fbADSREAD(			PORT						:= 500, 
					IDXGRP						:= udiIDXGRP_OFFS + nAxisID, 
					IDXOFFS						:= nOffset, 
					LEN							:= 2, 
					DESTADDR					:= ADR(wData), 
					READ						:= bExecute, 
					BUSY						=> Out.Busy, 
					ERR							=> Out.Error, 
					ERRID						=> Out.ErrorID);

// Fix library issue, one extra cycle + Done
CASE nStep OF
	
	0: 
	
		Out.Error 								:= FALSE;
		Out.ErrorID 							:= 0;

		IF Out.Busy THEN
			nStep								:= nStep + 10;
		END_IF
	
	10:
	
		IF NOT Out.Busy THEN
			Out.Busy							:= TRUE;
			IF Out.Error THEN
				Out.ErrorID						:= 0;
				Out.Error						:= FALSE;
				nStep							:= 1000;
			ELSE
				nStep							:= 100;
			END_IF
		END_IF
		
	100, 1000:

		Out.Done								:= nStep = 100;
		Out.Error								:= nStep = 1000;
		IF Out.Error THEN
			Message := CONCAT('FB_NcSWLimitSwitchCtrl method ReadBool failed - Error ID: ',UDINT_TO_STRING(Out.ErrorID));
			Message := CONCAT(Message, '! FB instance: %s');
			ADSLOGSTR(ADSLOG_MSGTYPE_WARN,Message,sInstancePath);
		END_IF
		
		IF bExecute THEN
			nStep								:= nStep + 1;
		ELSE
			fbADSREAD(	READ					:= FALSE);
			nStep								:= 0;
		END_IF
		
	101, 1001:
	
		Out.Done								:= nStep = 101;
		Out.Error								:= nStep = 1001;
		IF NOT bExecute THEN
			fbADSREAD(	READ					:= FALSE);
			Out.Done							:= FALSE;
			Out.Error							:= FALSE;
			Out.ErrorID							:= 0;
			nStep								:= 0;
		END_IF	

END_CASE

pRead											:= Out;

bOut											:= wData.0;
ReadBool										:= Out;
END_METHOD

METHOD ReadLreal 								: Tc2_MC2.ST_McOutputs
VAR_INPUT
	bExecute									: BOOL;
	nAxisID										: UDINT;
	nOffset										: UDINT;
END_VAR
VAR_OUTPUT
	lrOut										: LREAL;
END_VAR
VAR_INST
	fbADSREAD									: ADSREAD;
	lrData										: LREAL;
	nStep										: DINT;
END_VAR
VAR
	Out											: Tc2_MC2.ST_McOutputs;
	Message										: STRING;
END_VAR
IF nAxisID = 0 THEN
	
	IF NOT bAxisIdError THEN
		ADSLOGSTR(ADSLOG_MSGTYPE_ERROR,'FB_NcSWLimitSwitchCtrl critical error - Axis ID not assigned! FB instance: %s',sInstancePath);
	END_IF
	
	bAxisIdError 								:= TRUE;
	RETURN;	
END_IF

fbADSREAD(			PORT						:= 500, 
					IDXGRP						:= udiIDXGRP_OFFS + nAxisID, 
					IDXOFFS						:= nOffset, 
					LEN							:= 8, 
					DESTADDR					:= ADR(lrData), 
					READ						:= bExecute, 
					BUSY						=> Out.Busy, 
					ERR							=> Out.Error, 
					ERRID						=> Out.ErrorID);

// Fix library issue, one extra cycle + Done
CASE nStep OF
	
	0: 
	
		Out.Error 								:= FALSE;
		Out.ErrorID 							:= 0;

		IF Out.Busy THEN
			nStep								:= nStep + 10;
		END_IF
	
	10:
	
		IF NOT Out.Busy THEN
			Out.Busy							:= TRUE;
			IF Out.Error THEN
				Out.ErrorID						:= 0;
				Out.Error						:= FALSE;
				nStep							:= 1000;
			ELSE
				nStep							:= 100;
			END_IF
		END_IF
		
	100, 1000:

		Out.Done								:= nStep = 100;
		Out.Error								:= nStep = 1000;
		IF Out.Error THEN
			Message := CONCAT('FB_NcSWLimitSwitchCtrl method ReadLreal failed - Error ID: ',UDINT_TO_STRING(Out.ErrorID));
			Message := CONCAT(Message, '! FB instance: %s');
			ADSLOGSTR(ADSLOG_MSGTYPE_WARN,Message,sInstancePath);
		END_IF
		
		IF bExecute THEN
			nStep								:= nStep + 1;
		ELSE
			fbADSREAD(	READ					:= FALSE);
			nStep								:= 0;
		END_IF
		
	101, 1001:
	
		Out.Done								:= nStep = 101;
		Out.Error								:= nStep = 1001;
		IF NOT bExecute THEN
			fbADSREAD(	READ					:= FALSE);
			Out.Done							:= FALSE;
			Out.Error							:= FALSE;
			Out.ErrorID							:= 0;
			nStep								:= 0;
		END_IF	

END_CASE

pRead											:= Out;

lrOut											:= lrData;
ReadLreal										:= Out;
END_METHOD

METHOD ReadParams 								: Tc2_MC2.ST_McOutputs
VAR_INPUT
	bExecute									: BOOL;
	nAxisID										: UDINT;
END_VAR
VAR_INST
	stOut	 									: Tc2_MC2.ST_McOutputs;
	nStep										: DINT;
END_VAR
VAR
	Out	 										: Tc2_MC2.ST_McOutputs;
END_VAR
CASE nStep OF

	0: 
		IF bExecute THEN
			stOut.Busy							:= TRUE;
			nStep								:= nStep + 5;
		END_IF
		
	5:

		Out 									:= ReadValueMin(bExecute := TRUE, nAxisID := nAxisID);
		IF Out.Busy THEN
			nStep								:= nStep + 5;
		END_IF
	
	10:
	
		Out 									:= ReadValueMin(bExecute := FALSE, nAxisID := nAxisID);
		IF Out.Done THEN
			nStep								:= nStep + 5;
		ELSIF Out.Error THEN
			nStep								:= 1000;
		END_IF
	
	15: 
	
		Out 									:= ReadValueMax(bExecute := TRUE, nAxisID := nAxisID);
		IF Out.Busy THEN
			nStep								:= nStep + 5;
		END_IF
		
	20:
	
		Out 									:= ReadValueMax(bExecute := FALSE, nAxisID := nAxisID);
		IF Out.Done THEN
			nStep								:= nStep + 5;
		ELSIF Out.Error THEN
			nStep								:= 1000;
		END_IF
	
	25: 
	
		Out 									:= ReadStateMin(bExecute := TRUE, nAxisID := nAxisID);
		IF Out.Busy THEN
			nStep								:= nStep + 5;
		END_IF
		
	30:
	
		Out 									:= ReadStateMin(bExecute := FALSE, nAxisID := nAxisID);
		IF Out.Done THEN
			nStep								:= nStep + 5;
		ELSIF Out.Error THEN
			nStep								:= 1000;
		END_IF
	
	35: 
	
		Out 									:= ReadStateMax(bExecute := TRUE, nAxisID := nAxisID);
		IF Out.Busy THEN
			nStep								:= nStep + 5;
		END_IF
		
	40:
	
		Out 									:= ReadStateMax(bExecute := FALSE, nAxisID := nAxisID);
		IF Out.Done THEN
			nStep								:= 100;
		ELSIF Out.Error THEN
			nStep								:= 1000;
		END_IF
		
	100, 1000:

		stOut.Busy								:= FALSE;
		stOut.Done								:= nStep = 100;
		stOut.Error								:= nStep = 1000;
		nStep									:= nStep + 1;
		
	101, 1001:
	
		IF NOT bExecute THEN
			stOut.Busy							:= FALSE;
			stOut.Done							:= FALSE;
			stOut.Error							:= FALSE;
			nStep								:= 0;			
		END_IF

END_CASE

ReadParams										:= stOut;
END_METHOD

METHOD ReadStateMax 							: Tc2_MC2.ST_McOutputs
VAR_INPUT
	bExecute									: BOOL;
	nAxisID										: UDINT;
END_VAR
VAR
	bOut										: BOOL;
END_VAR
ReadStateMax 									:= ReadBool(	bExecute 	:= bExecute, 
																nAxisID 	:= nAxisID, 
																nOffset 	:= 16#0000_000C, 
																bOut 		=> bOut);

LimitSwitchStateMax								:= bOut;
END_METHOD

METHOD ReadStateMin 							: Tc2_MC2.ST_McOutputs
VAR_INPUT
	bExecute									: BOOL;
	nAxisID										: UDINT;
END_VAR
VAR
	bOut										: BOOL;
END_VAR
ReadStateMin 									:= ReadBool(	bExecute 	:= bExecute, 
																nAxisID 	:= nAxisID, 
																nOffset 	:= 16#0000_000B, 
																bOut 		=> bOut);
																
LimitSwitchStateMin								:= bOut;
END_METHOD

METHOD ReadValueMax 							: Tc2_MC2.ST_McOutputs
VAR_INPUT
	bExecute									: BOOL;
	nAxisID										: UDINT;
END_VAR
VAR
	lrOut										: LREAL;
END_VAR
ReadValueMax 									:= ReadLreal(	bExecute 	:= bExecute, 
																nAxisID 	:= nAxisID, 
																nOffset 	:= 16#0000_000E, 
																lrOut 		=> lrOut);
																
LimitSwitchPositionMax							:= lrOut;
END_METHOD

METHOD ReadValueMin 							: Tc2_MC2.ST_McOutputs
VAR_INPUT
	bExecute									: BOOL;
	nAxisID										: UDINT;
END_VAR
VAR
	lrOut										: LREAL;
END_VAR
ReadValueMin 									:= ReadLreal(	bExecute 	:= bExecute, 
																nAxisID 	:= nAxisID, 
																nOffset 	:= 16#0000_000D, 
																lrOut 		=> lrOut);
																
LimitSwitchPositionMin							:= lrOut;
END_METHOD

METHOD WriteBool 								: Tc2_MC2.ST_McOutputs
VAR_INPUT
	bExecute									: BOOL;
	bValue										: BOOL;
	nAxisID										: UDINT;
	nOffset										: UDINT;
END_VAR
VAR_INST
	fbADSWRITE									: ADSWRITE;
	wData										: WORD;
	nStep										: DINT;
END_VAR
VAR
	Out											: Tc2_MC2.ST_McOutputs;
	Message										: STRING;
END_VAR
IF nAxisID = 0 THEN
	
	IF NOT bAxisIdError THEN
		ADSLOGSTR(ADSLOG_MSGTYPE_ERROR,'FB_NcSWLimitSwitchCtrl critical error - Axis ID not assigned! FB instance: %s',sInstancePath);
	END_IF
	
	bAxisIdError 								:= TRUE;
	RETURN;	
END_IF

wData.0 										:= bValue;

fbADSWRITE(			PORT						:= 500, 
					IDXGRP						:= udiIDXGRP_OFFS + nAxisID, 
					IDXOFFS						:= nOffset, 
					LEN							:= 2, 
					SRCADDR						:= ADR(wData), 
					WRITE						:= bExecute, 
					BUSY						=> Out.Busy, 
					ERR							=> Out.Error, 
					ERRID						=> Out.ErrorID);

// Fix library issue, one extra cycle + Done
CASE nStep OF
	
	0: 
	
		Out.Error 								:= FALSE;
		Out.ErrorID 							:= 0;

		IF Out.Busy THEN
			nStep								:= nStep + 10;
		END_IF
	
	10:
	
		IF NOT Out.Busy THEN
			Out.Busy							:= TRUE;
			IF Out.Error THEN
				Out.ErrorID						:= 0;
				Out.Error						:= FALSE;
				nStep							:= 1000;
			ELSE
				nStep							:= 100;
			END_IF
		END_IF
		
	100, 1000:

		Out.Done								:= nStep = 100;
		Out.Error								:= nStep = 1000;
		IF Out.Error THEN
			Message := CONCAT('FB_NcSWLimitSwitchCtrl method WriteBool failed - Error ID: ',UDINT_TO_STRING(Out.ErrorID));
			Message := CONCAT(Message, '! FB instance: %s');
			ADSLOGSTR(ADSLOG_MSGTYPE_WARN,Message,sInstancePath);
		END_IF
		
		IF bExecute THEN
			nStep								:= nStep + 1;
		ELSE
			fbADSWRITE(	WRITE					:= FALSE);
			nStep								:= 0;
		END_IF
		
	101, 1001:
	
		Out.Done								:= nStep = 101;
		Out.Error								:= nStep = 1001;
		IF NOT bExecute THEN
			fbADSWRITE(	WRITE					:= FALSE);
			Out.Done							:= FALSE;
			Out.Error							:= FALSE;
			Out.ErrorID							:= 0;
			nStep								:= 0;
		END_IF	

END_CASE

pWrite											:= Out;
WriteBool										:= Out;
END_METHOD

METHOD WriteLreal 								: Tc2_MC2.ST_McOutputs
VAR_INPUT
	bExecute									: BOOL;
	lrValue										: LREAL;
	nAxisID										: UDINT;
	nOffset										: UDINT;
END_VAR
VAR_INST
	fbADSWRITE									: ADSWRITE;
	nStep										: DINT;
END_VAR
VAR
	Out											: Tc2_MC2.ST_McOutputs;
	Message										: STRING;
END_VAR
IF nAxisID = 0 THEN
	
	IF NOT bAxisIdError THEN
		ADSLOGSTR(ADSLOG_MSGTYPE_ERROR,'FB_NcSWLimitSwitchCtrl critical error - Axis ID not assigned! FB instance: %s',sInstancePath);
	END_IF
	
	bAxisIdError 								:= TRUE;
	RETURN;	
END_IF

fbADSWRITE(			PORT						:= 500, 
					IDXGRP						:= udiIDXGRP_OFFS + nAxisID, 
					IDXOFFS						:= nOffset, 
					LEN							:= 8, 
					SRCADDR						:= ADR(lrValue), 
					WRITE						:= bExecute, 
					BUSY						=> Out.Busy, 
					ERR							=> Out.Error, 
					ERRID						=> Out.ErrorID);

// Fix library issue, one extra cycle + Done
CASE nStep OF
	
	0: 
	
		Out.Error 								:= FALSE;
		Out.ErrorID 							:= 0;

		IF Out.Busy THEN
			nStep								:= nStep + 10;
		END_IF
	
	10:
	
		IF NOT Out.Busy THEN
			Out.Busy							:= TRUE;
			IF Out.Error THEN
				Out.ErrorID						:= 0;
				Out.Error						:= FALSE;
				nStep							:= 1000;
			ELSE
				nStep							:= 100;
			END_IF
		END_IF
		
	100, 1000:

		Out.Done								:= nStep = 100;
		Out.Error								:= nStep = 1000;
		IF Out.Error THEN
			Message := CONCAT('FB_NcSWLimitSwitchCtrl method WriteLreal failed - Error ID: ',UDINT_TO_STRING(Out.ErrorID));
			Message := CONCAT(Message, '! FB instance: %s');
			ADSLOGSTR(ADSLOG_MSGTYPE_WARN,Message,sInstancePath);
		END_IF
		
		IF bExecute THEN
			nStep								:= nStep + 1;
		ELSE
			fbADSWRITE(	WRITE					:= FALSE);
			nStep								:= 0;
		END_IF
		
	101, 1001:
	
		Out.Done								:= nStep = 101;
		Out.Error								:= nStep = 1001;
		IF NOT bExecute THEN
			fbADSWRITE(	WRITE					:= FALSE);
			Out.Done							:= FALSE;
			Out.Error							:= FALSE;
			Out.ErrorID							:= 0;
			nStep								:= 0;
		END_IF	

END_CASE

pWrite											:= Out;
WriteLreal										:= Out;
END_METHOD

METHOD WriteParams 								: Tc2_MC2.ST_McOutputs
VAR_INPUT
	bExecute									: BOOL;
	nAxisID										: UDINT;
END_VAR
VAR_INST
	stOut	 									: Tc2_MC2.ST_McOutputs;
	nStep										: DINT;
	lrLimitSwitchPositionMin					: LREAL 		:= 0;
	lrLimitSwitchPositionMax					: LREAL 		:= 0;
	bLimitSwitchStateMin						: BOOL 			:= FALSE;
	bLimitSwitchStateMax						: BOOL 			:= FALSE;
END_VAR
VAR
	Out	 										: Tc2_MC2.ST_McOutputs;
END_VAR
CASE nStep OF

	0: 
		IF bExecute THEN
			lrLimitSwitchPositionMin			:= LimitSwitchPositionMin;
			lrLimitSwitchPositionMax			:= LimitSwitchPositionMax;
			bLimitSwitchStateMin				:= LimitSwitchStateMin;
			bLimitSwitchStateMax				:= LimitSwitchStateMax;
			stOut.Busy							:= TRUE;
			nStep								:= nStep + 5;
		END_IF
		
	5:

		LimitSwitchPositionMin					:= lrLimitSwitchPositionMin;
		Out 									:= WriteValueMin(bExecute := TRUE, nAxisID := nAxisID);
		IF Out.Busy THEN
			nStep								:= nStep + 5;
		END_IF
	
	10:
	
		Out 									:= WriteValueMin(bExecute := FALSE, nAxisID := nAxisID);
		IF Out.Done THEN
			nStep								:= nStep + 5;
		ELSIF Out.Error THEN
			nStep								:= 1000;
		END_IF
	
	15: 
	
		LimitSwitchPositionMax					:= lrLimitSwitchPositionMax;
		Out 									:= WriteValueMax(bExecute := TRUE, nAxisID := nAxisID);
		IF Out.Busy THEN
			nStep								:= nStep + 5;
		END_IF
		
	20:
	
		Out 									:= WriteValueMax(bExecute := FALSE, nAxisID := nAxisID);
		IF Out.Done THEN
			nStep								:= nStep + 5;
		ELSIF Out.Error THEN
			nStep								:= 1000;
		END_IF
	
	25: 
	
		LimitSwitchStateMin						:= bLimitSwitchStateMin;
		Out 									:= WriteStateMin(bExecute := TRUE, nAxisID := nAxisID);
		IF Out.Busy THEN
			nStep								:= nStep + 5;
		END_IF
		
	30:
	
		Out 									:= WriteStateMin(bExecute := FALSE, nAxisID := nAxisID);
		IF Out.Done THEN
			nStep								:= nStep + 5;
		ELSIF Out.Error THEN
			nStep								:= 1000;
		END_IF
	
	35: 

		LimitSwitchStateMax						:= bLimitSwitchStateMax;	
		Out 									:= WriteStateMax(bExecute := TRUE, nAxisID := nAxisID);
		IF Out.Busy THEN
			nStep								:= nStep + 5;
		END_IF
		
	40:
	
		Out 									:= WriteStateMax(bExecute := FALSE, nAxisID := nAxisID);
		IF Out.Done THEN
			nStep								:= 100;
		ELSIF Out.Error THEN
			nStep								:= 1000;
		END_IF
		
	100, 1000:

		stOut.Busy								:= FALSE;
		stOut.Done								:= nStep = 100;
		stOut.Error								:= nStep = 1000;
		nStep									:= nStep + 1;
		
	101, 1001:
	
		IF NOT bExecute THEN
			stOut.Busy							:= FALSE;
			stOut.Done							:= FALSE;
			stOut.Error							:= FALSE;
			nStep								:= 0;			
		END_IF

END_CASE

WriteParams										:= stOut;
END_METHOD

METHOD WriteStateMax 							: Tc2_MC2.ST_McOutputs
VAR_INPUT
	bExecute									: BOOL;
	nAxisID										: UDINT;
END_VAR
WriteStateMax 									:= WriteBool(	bExecute 	:= bExecute,
 																bValue		:= LimitSwitchStateMax,
																nAxisID 	:= nAxisID, 
																nOffset 	:= 16#0000_000C);
END_METHOD

METHOD WriteStateMin 							: Tc2_MC2.ST_McOutputs
VAR_INPUT
	bExecute									: BOOL;
	nAxisID										: UDINT;
END_VAR
WriteStateMin 									:= WriteBool(	bExecute 	:= bExecute,
 																bValue		:= LimitSwitchStateMin,
																nAxisID 	:= nAxisID, 
																nOffset 	:= 16#0000_000B);
END_METHOD

METHOD WriteValueMax 							: Tc2_MC2.ST_McOutputs
VAR_INPUT
	bExecute									: BOOL;
	nAxisID										: UDINT;
END_VAR
WriteValueMax 									:= WriteLreal(	bExecute 	:= bExecute, 
																lrValue		:= LimitSwitchPositionMax,
																nAxisID 	:= nAxisID, 
																nOffset 	:= 16#0000_000E);
END_METHOD

METHOD WriteValueMin 							: Tc2_MC2.ST_McOutputs
VAR_INPUT
	bExecute									: BOOL;
	nAxisID										: UDINT;
END_VAR
WriteValueMin 									:=  WriteLreal(	bExecute 	:= bExecute, 
																lrValue		:= LimitSwitchPositionMin,
																nAxisID 	:= nAxisID, 
																nOffset 	:= 16#0000_000D);
END_METHOD

END_FUNCTION_BLOCK

// ---- POUs/FB/AxisControl/Internal/FB_NcPosLagMonitoring.TcPOU
//==================================================================================================
//							Beckhoff Automation Poland
//									03.01.2023
//
// Code owner: TG
//
// Sample code to maitenance software limit switches
//
// Used libraries: 
//	Tc2_MC2							|| 3.3.48.0
//	Tc2_System						|| 3.4.26.0
//
//
// 	v1.0 	|| TC v 3.1.4024.35 	|| First edition
//==================================================================================================
{attribute 'reflection'}
FUNCTION_BLOCK FB_NcPosLagMonitoring
VAR CONSTANT
	udiIDXGRP_OFFS								: UDINT := 16#0000_6000;
END_VAR
VAR
	{attribute 'instance-path'}
	{attribute 'noinit'}
	sInstancePath								: STRING;

	_stRead										: Tc2_MC2.ST_McOutputs;
	_stWrite									: Tc2_MC2.ST_McOutputs;
	_fValue										: LREAL 		:= 0;
	_bState										: BOOL 			:= FALSE;
	bAxisIdError								: BOOL;
END_VAR

PROPERTY bState 					: BOOL
GET
bState											:= _bState;
END_GET
SET
_bState											:= bState;
END_SET
END_PROPERTY

PROPERTY fValue 				: LREAL
GET
fValue											:= _fValue;
END_GET
SET
_fValue											:= fValue;
END_SET
END_PROPERTY

PROPERTY pRead 							: Tc2_MC2.ST_McOutputs
GET
pRead											:= _stRead;
END_GET
SET
_stRead											:= pRead;
END_SET
END_PROPERTY

PROPERTY pWrite 							: Tc2_MC2.ST_McOutputs
GET
pWrite											:= _stWrite;
END_GET
SET
_stWrite										:= pWrite;
END_SET
END_PROPERTY

// Needs one cycle extra with false execution, after busy false
METHOD ReadBool 								: Tc2_MC2.ST_McOutputs
VAR_INPUT
	bExecute									: BOOL;
	nAxisID										: UDINT;
	nOffset										: UDINT;
END_VAR
VAR_OUTPUT
	bOut										: BOOL;
END_VAR
VAR_INST
	fbADSREAD									: ADSREAD;
	wData										: WORD;
	nStep										: DINT;
END_VAR
VAR
	Out											: Tc2_MC2.ST_McOutputs;
	Message										: STRING;
END_VAR
IF nAxisID = 0 THEN
	
	IF NOT bAxisIdError THEN
		ADSLOGSTR(ADSLOG_MSGTYPE_ERROR,'FB_NcSWLimitSwitchCtrl critical error - Axis ID not assigned! FB instance: %s',sInstancePath);
	END_IF
	
	bAxisIdError 								:= TRUE;
	RETURN;	
END_IF

fbADSREAD(			PORT						:= 500, 
					IDXGRP						:= udiIDXGRP_OFFS + nAxisID, 
					IDXOFFS						:= nOffset, 
					LEN							:= 2, 
					DESTADDR					:= ADR(wData), 
					READ						:= bExecute, 
					BUSY						=> Out.Busy, 
					ERR							=> Out.Error, 
					ERRID						=> Out.ErrorID);

// Fix library issue, one extra cycle + Done
CASE nStep OF
	
	0: 
	
		Out.Error 								:= FALSE;
		Out.ErrorID 							:= 0;

		IF Out.Busy THEN
			nStep								:= nStep + 10;
		END_IF
	
	10:
	
		IF NOT Out.Busy THEN
			Out.Busy							:= TRUE;
			IF Out.Error THEN
				Out.ErrorID						:= 0;
				Out.Error						:= FALSE;
				nStep							:= 1000;
			ELSE
				nStep							:= 100;
			END_IF
		END_IF
		
	100, 1000:

		Out.Done								:= nStep = 100;
		Out.Error								:= nStep = 1000;
		IF Out.Error THEN
			Message := CONCAT('FB_NcSWLimitSwitchCtrl method ReadBool failed - Error ID: ',UDINT_TO_STRING(Out.ErrorID));
			Message := CONCAT(Message, '! FB instance: %s');
			ADSLOGSTR(ADSLOG_MSGTYPE_WARN,Message,sInstancePath);
		END_IF
		
		IF bExecute THEN
			nStep								:= nStep + 1;
		ELSE
			fbADSREAD(	READ					:= FALSE);
			nStep								:= 0;
		END_IF
		
	101, 1001:
	
		Out.Done								:= nStep = 101;
		Out.Error								:= nStep = 1001;
		IF NOT bExecute THEN
			fbADSREAD(	READ					:= FALSE);
			Out.Done							:= FALSE;
			Out.Error							:= FALSE;
			Out.ErrorID							:= 0;
			nStep								:= 0;
		END_IF	

END_CASE

pRead											:= Out;

bOut											:= wData.0;
ReadBool										:= Out;
END_METHOD

METHOD ReadLreal 								: Tc2_MC2.ST_McOutputs
VAR_INPUT
	bExecute									: BOOL;
	nAxisID										: UDINT;
	nOffset										: UDINT;
END_VAR
VAR_OUTPUT
	lrOut										: LREAL;
END_VAR
VAR_INST
	fbADSREAD									: ADSREAD;
	lrData										: LREAL;
	nStep										: DINT;
END_VAR
VAR
	Out											: Tc2_MC2.ST_McOutputs;
	Message										: STRING;
END_VAR
IF nAxisID = 0 THEN
	
	IF NOT bAxisIdError THEN
		ADSLOGSTR(ADSLOG_MSGTYPE_ERROR,'FB_NcSWLimitSwitchCtrl critical error - Axis ID not assigned! FB instance: %s',sInstancePath);
	END_IF
	
	bAxisIdError 								:= TRUE;
	RETURN;	
END_IF

fbADSREAD(			PORT						:= 500, 
					IDXGRP						:= udiIDXGRP_OFFS + nAxisID, 
					IDXOFFS						:= nOffset, 
					LEN							:= 8, 
					DESTADDR					:= ADR(lrData), 
					READ						:= bExecute, 
					BUSY						=> Out.Busy, 
					ERR							=> Out.Error, 
					ERRID						=> Out.ErrorID);

// Fix library issue, one extra cycle + Done
CASE nStep OF
	
	0: 
	
		Out.Error 								:= FALSE;
		Out.ErrorID 							:= 0;

		IF Out.Busy THEN
			nStep								:= nStep + 10;
		END_IF
	
	10:
	
		IF NOT Out.Busy THEN
			Out.Busy							:= TRUE;
			IF Out.Error THEN
				Out.ErrorID						:= 0;
				Out.Error						:= FALSE;
				nStep							:= 1000;
			ELSE
				nStep							:= 100;
			END_IF
		END_IF
		
	100, 1000:

		Out.Done								:= nStep = 100;
		Out.Error								:= nStep = 1000;
		IF Out.Error THEN
			Message := CONCAT('FB_NcSWLimitSwitchCtrl method ReadLreal failed - Error ID: ',UDINT_TO_STRING(Out.ErrorID));
			Message := CONCAT(Message, '! FB instance: %s');
			ADSLOGSTR(ADSLOG_MSGTYPE_WARN,Message,sInstancePath);
		END_IF
		
		IF bExecute THEN
			nStep								:= nStep + 1;
		ELSE
			fbADSREAD(	READ					:= FALSE);
			nStep								:= 0;
		END_IF
		
	101, 1001:
	
		Out.Done								:= nStep = 101;
		Out.Error								:= nStep = 1001;
		IF NOT bExecute THEN
			fbADSREAD(	READ					:= FALSE);
			Out.Done							:= FALSE;
			Out.Error							:= FALSE;
			Out.ErrorID							:= 0;
			nStep								:= 0;
		END_IF	

END_CASE

pRead											:= Out;

lrOut											:= lrData;
ReadLreal										:= Out;
END_METHOD

METHOD ReadState 								: Tc2_MC2.ST_McOutputs
VAR_INPUT
	bExecute									: BOOL;
	nAxisID										: UDINT;
END_VAR
VAR
	bOut										: BOOL;
END_VAR
ReadState 										:= ReadBool(	bExecute 	:= bExecute, 
																nAxisID 	:= nAxisID, 
																nOffset 	:= 16#0000_0010, 
																bOut 		=> bOut);

bState											:= bOut;
END_METHOD

METHOD ReadValue 								: Tc2_MC2.ST_McOutputs
VAR_INPUT
	bExecute									: BOOL;
	nAxisID										: UDINT;
END_VAR
VAR
	lrOut										: LREAL;
END_VAR
ReadValue 										:= ReadLreal(	bExecute 	:= bExecute, 
																nAxisID 	:= nAxisID, 
																nOffset 	:= 16#0000_0012, 
																lrOut 		=> lrOut);
																
fValue											:= lrOut;
END_METHOD

METHOD WriteBool 								: Tc2_MC2.ST_McOutputs
VAR_INPUT
	bExecute									: BOOL;
	bValue										: BOOL;
	nAxisID										: UDINT;
	nOffset										: UDINT;
END_VAR
VAR_INST
	fbADSWRITE									: ADSWRITE;
	wData										: WORD;
	nStep										: DINT;
END_VAR
VAR
	Out											: Tc2_MC2.ST_McOutputs;
	Message										: STRING;
END_VAR
IF nAxisID = 0 THEN
	
	IF NOT bAxisIdError THEN
		ADSLOGSTR(ADSLOG_MSGTYPE_ERROR,'FB_NcSWLimitSwitchCtrl critical error - Axis ID not assigned! FB instance: %s',sInstancePath);
	END_IF
	
	bAxisIdError 								:= TRUE;
	RETURN;	
END_IF

wData.0 										:= bValue;

fbADSWRITE(			PORT						:= 500, 
					IDXGRP						:= udiIDXGRP_OFFS + nAxisID, 
					IDXOFFS						:= nOffset, 
					LEN							:= 2, 
					SRCADDR						:= ADR(wData), 
					WRITE						:= bExecute, 
					BUSY						=> Out.Busy, 
					ERR							=> Out.Error, 
					ERRID						=> Out.ErrorID);

// Fix library issue, one extra cycle + Done
CASE nStep OF
	
	0: 
	
		Out.Error 								:= FALSE;
		Out.ErrorID 							:= 0;

		IF Out.Busy THEN
			nStep								:= nStep + 10;
		END_IF
	
	10:
	
		IF NOT Out.Busy THEN
			Out.Busy							:= TRUE;
			IF Out.Error THEN
				Out.ErrorID						:= 0;
				Out.Error						:= FALSE;
				nStep							:= 1000;
			ELSE
				nStep							:= 100;
			END_IF
		END_IF
		
	100, 1000:

		Out.Done								:= nStep = 100;
		Out.Error								:= nStep = 1000;
		IF Out.Error THEN
			Message := CONCAT('FB_NcSWLimitSwitchCtrl method WriteBool failed - Error ID: ',UDINT_TO_STRING(Out.ErrorID));
			Message := CONCAT(Message, '! FB instance: %s');
			ADSLOGSTR(ADSLOG_MSGTYPE_WARN,Message,sInstancePath);
		END_IF
		
		IF bExecute THEN
			nStep								:= nStep + 1;
		ELSE
			fbADSWRITE(	WRITE					:= FALSE);
			nStep								:= 0;
		END_IF
		
	101, 1001:
	
		Out.Done								:= nStep = 101;
		Out.Error								:= nStep = 1001;
		IF NOT bExecute THEN
			fbADSWRITE(	WRITE					:= FALSE);
			Out.Done							:= FALSE;
			Out.Error							:= FALSE;
			Out.ErrorID							:= 0;
			nStep								:= 0;
		END_IF	

END_CASE

pWrite											:= Out;
WriteBool										:= Out;
END_METHOD

METHOD WriteLreal 								: Tc2_MC2.ST_McOutputs
VAR_INPUT
	bExecute									: BOOL;
	lrValue										: LREAL;
	nAxisID										: UDINT;
	nOffset										: UDINT;
END_VAR
VAR_INST
	fbADSWRITE									: ADSWRITE;
	nStep										: DINT;
END_VAR
VAR
	Out											: Tc2_MC2.ST_McOutputs;
	Message										: STRING;
END_VAR
IF nAxisID = 0 THEN
	
	IF NOT bAxisIdError THEN
		ADSLOGSTR(ADSLOG_MSGTYPE_ERROR,'FB_NcSWLimitSwitchCtrl critical error - Axis ID not assigned! FB instance: %s',sInstancePath);
	END_IF
	
	bAxisIdError 								:= TRUE;
	RETURN;	
END_IF

fbADSWRITE(			PORT						:= 500, 
					IDXGRP						:= udiIDXGRP_OFFS + nAxisID, 
					IDXOFFS						:= nOffset, 
					LEN							:= 8, 
					SRCADDR						:= ADR(lrValue), 
					WRITE						:= bExecute, 
					BUSY						=> Out.Busy, 
					ERR							=> Out.Error, 
					ERRID						=> Out.ErrorID);

// Fix library issue, one extra cycle + Done
CASE nStep OF
	
	0: 
	
		Out.Error 								:= FALSE;
		Out.ErrorID 							:= 0;

		IF Out.Busy THEN
			nStep								:= nStep + 10;
		END_IF
	
	10:
	
		IF NOT Out.Busy THEN
			Out.Busy							:= TRUE;
			IF Out.Error THEN
				Out.ErrorID						:= 0;
				Out.Error						:= FALSE;
				nStep							:= 1000;
			ELSE
				nStep							:= 100;
			END_IF
		END_IF
		
	100, 1000:

		Out.Done								:= nStep = 100;
		Out.Error								:= nStep = 1000;
		IF Out.Error THEN
			Message := CONCAT('FB_NcSWLimitSwitchCtrl method WriteLreal failed - Error ID: ',UDINT_TO_STRING(Out.ErrorID));
			Message := CONCAT(Message, '! FB instance: %s');
			ADSLOGSTR(ADSLOG_MSGTYPE_WARN,Message,sInstancePath);
		END_IF
		
		IF bExecute THEN
			nStep								:= nStep + 1;
		ELSE
			fbADSWRITE(	WRITE					:= FALSE);
			nStep								:= 0;
		END_IF
		
	101, 1001:
	
		Out.Done								:= nStep = 101;
		Out.Error								:= nStep = 1001;
		IF NOT bExecute THEN
			fbADSWRITE(	WRITE					:= FALSE);
			Out.Done							:= FALSE;
			Out.Error							:= FALSE;
			Out.ErrorID							:= 0;
			nStep								:= 0;
		END_IF	

END_CASE

pWrite											:= Out;
WriteLreal										:= Out;
END_METHOD

METHOD WriteState 								: Tc2_MC2.ST_McOutputs
VAR_INPUT
	bExecute									: BOOL;
	nAxisID										: UDINT;
END_VAR
WriteState 										:= WriteBool(	bExecute 	:= bExecute,
 																bValue		:= bState,
																nAxisID 	:= nAxisID, 
																nOffset 	:= 16#0000_0010);
END_METHOD

METHOD WriteValue 								: Tc2_MC2.ST_McOutputs
VAR_INPUT
	bExecute									: BOOL;
	nAxisID										: UDINT;
END_VAR
WriteValue 										:= WriteLreal(	bExecute 	:= bExecute, 
																lrValue		:= fValue,
																nAxisID 	:= nAxisID, 
																nOffset 	:= 16#0000_0012);
END_METHOD

END_FUNCTION_BLOCK

// ---- POUs/FB/AxisControl/Internal/HomingAdv/FB_HomingTorqueDetection.TcPOU
//==================================================================================================
//							Beckhoff Automation Poland
//									3.01.2023
//	Function block running home procedure in torque mode detection
//	It doesn't change position - only detection implemented
//	lrRecordedPosition - catched position. Offset can be written i.e. to encoder memory
//
//	Avaliable two modes:
//	1. Lag based - bLagBased = TRUE - define lrLagLimit which decides about end of movement
//	2. Torque based - bLagBased = FALSE - define lrTorqueLimit and lrTorqueTolerance which decides about end of movement
//
//	Library: Tc3_MC2_AdvancedHoming, Tc2_MC2, 
//
//  v1.1	|| TC v 3.1.4024.35		|| Naming convention 
//  v1.0	|| TC v 3.1.4024.22		|| First edition 
//==================================================================================================
FUNCTION_BLOCK FB_HomingTorqueDetection
VAR_IN_OUT
	Axis 										: Tc2_MC2.AXIS_REF;
END_VAR  
VAR_INPUT
	bExecute									: BOOL;					// The command is executed with a rising edge.
	bLagBased									: BOOL;					// TRUE: MC_StepBlockLagBased, FALSE: MC_StepBlock
	eDirection									: Tc3_MC2_AdvancedHoming.MC_Home_Direction;	// 
	fVelocity									: LREAL;				// Maximum travel velocity (>0)
	fDetectionVelocityLimit						: LREAL;				// Velocity that must be fallen below for the time DetectionVelocityTime in order to detect driving against the fixed stop.
	tDetectionVelocityTime						: TIME;					// Time for detecting the velocity undershoot when driving against the fixed stop.
	tTimeLimit									: TIME;					// Exceeding this time leads to the search procedure being aborted.
	fDistanceLimit								: LREAL;				// Exceeding this distance in relation to the start position leads to the search procedure being aborted.
	fTorqueLimit								: LREAL;				// The motor torque is limited to this value, in relation to the weight counterbalance that is possibly parameterized in the drive, in order to avoid mechanical damage.
	fTorqueTolerance							: LREAL;				// Tolerance related to the TorqueLimit within which driving against the fixed stop is detected.
	fLagLimit									: LREAL;				// Position lag value which, if exceeded, leads to detection of driving against the fixed stop.
	fDistance									: LREAL;				// Distance by which the axis moves away from the current position.
END_VAR                             		
VAR_OUTPUT                              		
	bDone										: BOOL;
	bBusy										: BOOL;
	bCommandAborted								: BOOL;
	bError										: BOOL;
	nErrorID									: UDINT;
	fRecordedPosition							: LREAL;				// Catched position. Offset can be written i.e. to encoder memory
END_VAR
VAR
//=========================== Common ============================
	nStep										: DINT;
	stParameter									: Tc3_MC2_AdvancedHoming.MC_HomingParameter;
	stOptions									: Tc3_MC2_AdvancedHoming.ST_Home_Options3;
//========================= Step Block ==========================
	mcStepBlock									: Tc3_MC2_AdvancedHoming.MC_StepBlockDetection ;
	mcStepBlockLag								: Tc3_MC2_AdvancedHoming.MC_StepBlockLagBasedDetection;
//====================== Move Relative ==========================
	mcMoveRelative								: MC_MoveRelative;
//============================ Abort ============================
	mcAbortHoming								: Tc3_MC2_AdvancedHoming.MC_AbortHoming;
//========================== Internal ===========================
    {attribute 'hide'}
	nErrorID_Int								: UDINT;
//===============================================================
END_VAR

//====== Call FBs outside CASE - easier debugging ===============
mcStepBlockLag(Axis								:= Axis, 
				Parameter						:= stParameter);
				                        		
mcStepBlock(	Axis							:= Axis, 
				Parameter						:= stParameter);	

mcMoveRelative(	Axis							:= Axis);
                                        		
mcAbortHoming(	Axis							:= Axis, 
				Parameter						:= stParameter);
			
//============== CASE instruction - step machine ================
CASE nStep OF
	
	0: // Wait for command
	
		IF bExecute THEN
			bBusy								:= TRUE;
			// Latch finish parameters
			mcMoveRelative.Distance				:= fDistance;
			mcMoveRelative.Velocity				:= fVelocity;
			
			IF bLagBased THEN

				mcStepBlockLag(Axis				:= Axis, 
						Parameter				:= stParameter, 
						Execute					:= TRUE, 
						Direction				:= eDirection, 
						Velocity				:= fVelocity,
						DetectionVelocityLimit	:= fDetectionVelocityLimit, 
						DetectionVelocityTime	:= tDetectionVelocityTime, 
						TimeLimit				:= tTimeLimit, 
						DistanceLimit			:= fDistanceLimit, 
						TorqueLimit				:= fTorqueLimit, 
						LagLimit				:= fLagLimit, 
						Options					:= stOptions);
				
				nStep							:= 1000;
				
			ELSE

				mcStepBlock(Axis				:= Axis, 
						Parameter				:= stParameter, 
						Execute					:= TRUE, 
						Direction				:= eDirection, 
						Velocity				:= fVelocity,
						DetectionVelocityLimit	:= fDetectionVelocityLimit, 
						DetectionVelocityTime	:= tDetectionVelocityTime, 
						TimeLimit				:= tTimeLimit, 
						DistanceLimit			:= fDistanceLimit, 
						TorqueLimit				:= fTorqueLimit, 
						TorqueTolerance			:= fTorqueTolerance, 
						Options					:= stOptions);
						
				nStep							:= 2000;
				
			END_IF
		END_IF
	
	1000: // Wait till end MC_StepBlockLagBasedDetection
	
		IF mcStepBlockLag.Done THEN
			fRecordedPosition					:= mcStepBlockLag.RecordedPosition;
			mcStepBlockLag.Execute				:= FALSE;
			nStep 								:= 3000;
		END_IF
		
		IF mcStepBlockLag.CommandAborted THEN
			mcStepBlockLag.Execute				:= FALSE;
			nStep 								:= 6010;
		END_IF
		
		IF mcStepBlockLag.Error THEN
			mcStepBlockLag.Execute				:= FALSE;
			nErrorID_Int						:= mcStepBlockLag.ErrorID;
			nStep 								:= 6110;
		END_IF
	
	2000: // Wait till end MC_StepBlockDetection
	
		IF mcStepBlock.Done THEN
			fRecordedPosition					:= mcStepBlock.RecordedPosition;
			mcStepBlock.Execute					:= FALSE;
			nStep 								:= 3000;
		END_IF
		
		IF mcStepBlock.CommandAborted THEN
			mcStepBlock.Execute					:= FALSE;
			nStep 								:= 6020;
		END_IF
		
		IF mcStepBlock.Error THEN
			mcStepBlock.Execute					:= FALSE;
			nErrorID_Int						:= mcStepBlock.ErrorID;
			nStep 								:= 6120;
		END_IF
		
	3000:	// MC_AbortHoming - way of finish homing procedure
	
		mcAbortHoming.Execute					:= TRUE;				
		nStep									:= nStep + 10;
		
	3010: // Wait till end MC_HomeDirect
	
		IF mcAbortHoming.Done THEN
			mcAbortHoming.Execute				:= FALSE;
			nStep 								:= 4000;
		END_IF
		
		IF mcAbortHoming.CommandAborted THEN
			mcAbortHoming.Execute				:= FALSE;
			nStep 								:= 6040;
		END_IF
		
		IF mcAbortHoming.Error THEN
			mcAbortHoming.Execute				:= FALSE;
			nErrorID							:= mcAbortHoming.ErrorID;
			nStep 								:= 6140;
		END_IF		

	4000: // MC_MoveRelative
	
		mcMoveRelative.Execute					:= TRUE;			
		nStep									:= nStep + 10;
	
	4010: // Wait till end MC_MoveRelative
	
		IF mcMoveRelative.Done THEN
			mcMoveRelative.Execute				:= FALSE;
			bBusy 								:= FALSE;
			bDone 								:= TRUE;
			nStep								:= 5000;
		END_IF
		
		IF mcMoveRelative.CommandAborted THEN
			mcMoveRelative.Execute				:= FALSE;
			nStep 								:= 6050;
		END_IF
		
		IF mcMoveRelative.Error THEN
			mcMoveRelative.Execute				:= FALSE;
			nErrorID_Int						:= mcMoveRelative.ErrorID;
			nStep 								:= 6150;
		END_IF		
	
	5000: // Done
	
		bDone									:= bExecute;
		IF NOT bExecute THEN
			fRecordedPosition					:= 0;
			nStep 								:= 0;
		END_IF
	
	6000..6199: // MC_AbortHoming
	
		mcAbortHoming.Execute					:= TRUE;				
		nStep									:= nStep + 200;
	
	6200..6399: // Wait till end Command Aborted (..200-..299)/Error (..300/399)
	
		// No matter what is the end, we go to Command Aborted/Error State
		IF NOT mcAbortHoming.Busy THEN
			mcAbortHoming.Execute				:= FALSE;
			bBusy 								:= FALSE;
			// Set CA/E flag
			bCommandAborted						:= nStep < 6300;
			bError								:= NOT bCommandAborted;
			
			IF bError THEN
				nErrorID						:= nErrorID_Int;
				nStep							:= nStep + 10000;
			ELSE
				nStep							:= 7000;
			END_IF
		
		END_IF		
	
	7000: // Command Aborted
	
		bCommandAborted							:= bExecute;
		IF NOT bExecute THEN
			nStep 								:= 0;
		END_IF
		
	10000..20000: // Error
	
		bError									:= bExecute;
		IF NOT bExecute THEN
			nErrorID							:= 0;
			nErrorID_Int						:= 0;
			nStep 								:= 0;
		END_IF
		
END_CASE
//===============================================================

END_FUNCTION_BLOCK

// ---- POUs/FB/FB_DigitalInput_1.TcPOU
//==================================================================================================
//							Beckhoff Automation Poland
//									14.03.2023
//
// Code owner: TG
//
// Function block for processing digital inputs. 
// Includes filters, simulating and edges detection.
//
// Used libraries: 
//	Tc2_standard						|| 3.3.3.0
//
// Used FBs:
//
// Used DUTs:
//
//  v1.0	|| TC v 3.1.4024.40		|| First edition
//==================================================================================================
FUNCTION_BLOCK FB_DigitalInput_1

VAR_INPUT
	In 											: BOOL;
END_VAR

VAR
	
	bManual										: BOOL;	 // HMI
	bManualIn									: BOOL;	 // HMI
	{attribute 'hide'}
	_bCheckFS									: BOOL;
	{attribute 'hide'}
	_bIn	 									: BOOL;
	{attribute 'hide'}
	_bInRE										: BOOL;
	{attribute 'hide'}
	_bInFE										: BOOL;
	{attribute 'hide'}
	_tTimeOn									: TIME;
	{attribute 'hide'}
	_tTimeOff									: TIME;	
	{attribute 'hide'}
	_tTimeFS									: TIME;
	{attribute 'hide'}
	TimeFS										: TOF;	
	{attribute 'hide'}
	rtTrigger									: R_TRIG;
	{attribute 'hide'}
	ftTrigger									: F_TRIG;
END_VAR

{attribute 'monitoring' := 'variable'}
PROPERTY bCheckFS								: BOOL
GET
bCheckFS										:= _bCheckFS;
END_GET
SET
_bCheckFS										:= bCheckFS;
END_SET
END_PROPERTY

{attribute 'monitoring' := 'variable'}
PROPERTY bErrFS 								: BOOL							//Fail-safe error
GET
bErrFS											:= NOT TimeFS.Q AND bCheckFS;
END_GET
END_PROPERTY

{attribute 'monitoring' := 'variable'}
PROPERTY bIn 									: BOOL							//Processed input variable
GET
bIn												:= _bIn;
END_GET
SET
_bIn											:= bIn;
END_SET
END_PROPERTY

{attribute 'monitoring' := 'variable'}
PROPERTY bInFE 									: BOOL							//Falling edge detected
GET
bInFE											:= ftTrigger.Q;
END_GET
END_PROPERTY

{attribute 'monitoring' := 'variable'}
PROPERTY bInRE 									: BOOL							//Rising edge detected
GET
bInRE											:= rtTrigger.Q;
END_GET
END_PROPERTY

METHOD Filter 									: BOOL							//Activation and disable filter
VAR_INST
	{attribute 'hide'}
	TimeON										: TON;
	{attribute 'hide'}
	TimeOFF										: TOF;	
END_VAR
TimeON(IN := In, PT := tTimeON);
TimeOFF(IN := TimeON.Q, PT := tTimeOff);

bIn												:= TimeOFF.Q;
END_METHOD

METHOD FilterTrig 								: BOOL						//Activation and disable filter with edges detection
Filter();		
RTrig();
FTrig();
END_METHOD

METHOD FS 										: BOOL								// Fail-safe detection timer
VAR_INST
	{attribute 'hide'}
	bLastIn										: BOOL;	
END_VAR
TimeFS(IN := bLastIn <> In, PT := tTimeFS);	

bLastIn											:= In;
END_METHOD

METHOD PRIVATE FTrig 							: BOOL							// Falling edge detection
ftTrigger(CLK := bIn);
END_METHOD

METHOD Manual 									: BOOL							//Manually controlled input
IF bManual THEN
	ManualEx(bIn := bManualIn);
END_IF
END_METHOD

METHOD ManualEx 									: BOOL							//Manually controlled input
VAR_INPUT
	bIn												: BOOL;
END_VAR
bCheckFS										:= FALSE;
bIn												:= bIn;
END_METHOD

METHOD ManualExTrig 								: BOOL						//Manually controlled input with edges detection
VAR_INPUT
	bManual											: BOOL;
	bIn												: BOOL;
END_VAR
ManualEx(bIn := bManualIn);		
RTrig();
FTrig();
END_METHOD

METHOD ManualTrig 								: BOOL						//Manually controlled input with edges detection
Manual();		
RTrig();
FTrig();
END_METHOD

METHOD Raw 										: BOOL							// Raw value
bIn												:= In;
END_METHOD

METHOD PRIVATE RTrig 							: BOOL							//Rising edge detection
rtTrigger(CLK := bIn);
END_METHOD

{attribute 'monitoring' := 'variable'}
PROPERTY tTimeFS 								: TIME							//fail-safe control time [ms]
GET
tTimeFS											:= _tTimeFS;
END_GET
SET
_tTimeFS										:= tTimeFS;
END_SET
END_PROPERTY

{attribute 'monitoring' := 'variable'}
PROPERTY tTimeOff 								: TIME						//disabling filter time [ms]
GET
tTimeOff										:= _tTimeOff;
END_GET
SET
_tTimeOff										:= tTimeOff;
END_SET
END_PROPERTY

{attribute 'monitoring' := 'variable'}
PROPERTY tTimeOn 								: TIME							//activation delay time [ms]
GET
tTimeOn											:= _tTimeOn;
END_GET
SET
_tTimeOn									:= tTimeOn;
END_SET
END_PROPERTY

END_FUNCTION_BLOCK

// ---- POUs/Recipes/P030_Recipes.TcPOU
 PROGRAM P030_Recipes
 VAR_INPUT
	aRecipeListString									:	ARRAY[0..udiMaxRecipeCount] OF STRING(255);		//Recipes FROM/TO C:\Recipes\LIST.BIN
	aRecipeParamsVariables								:	ARRAY[0..udiMaxParamsVariablesCount-1] OF STRING(255);
	aRecipeParamsValues									:	ARRAY[0..udiMaxParamsVariablesCount-1] OF STRING(255);
 END_VAR

VAR

	//Edit
	wsEditOldCaption									:	WSTRING;
	udiEditNewIndex			:	UDINT;
	udiEditOldIndex			:	UDINT;
	wsEditNewCaption1		:	WSTRING:= "";
	wsEditNewCaption2		:	WSTRING:= "";
	bEditOk					:	BOOL;
	bEditFail				:	BOOL;
	wsEditErrorMessage		:	WSTRING;
	//end of Edit
	
	//zmiany Vasyl
	bRecipeLoaded										:BOOL;
	bRecipeDelete										:BOOL;
	bRecipeDeleteAck									:BOOL;                                                  	
	bCreateOrClone										:BOOL;	
	bRecipeEdit											:BOOL;	
	bRecipeShowEdit										:BOOL;	
	wsInfoNope											:WSTRING;
	bRecipeLoad											:BOOL;
	bRecipeLoadAck										:BOOL;
	tonCreateOrClone									:TON;
	
	fbRecipeLoad										:	FB_LoadCSV;									//FB for loading binary file
	fbRecipeSave										:	FB_RecipeSaveCSV;
	fbRecipeVariablesSave								:	FB_RecipeVariablesSaveCSV;
	sRecipeFilePath										:	STRING;	

	stActRecipe											:	ST_Recipe;	
	
	bInit												:	BOOL;
	
	//Wiska
	udiCurrentIndex			:	UDINT;
	wsCurrentCaption1		:	WSTRING:= "";
	wsCurrentCaption2		:	WSTRING:= "";	

	//Main user list
	aRecipeList											:	ARRAY[0..udiMaxRecipeCount] OF ST_RecipeListItem;		//Recipes FROM/TO C:\Recipes\LIST.BIN
	
	//Load & save operations
	udiInitCase											:	UDINT;										//Init case (load file or set default and save default
	udiUpdateCase										:	UDINT;										//Update file on HDD case
	fbListLoad											:	FB_LoadCSV;									//FB for loading binary file
	fbListSave											:	FB_ListSaveCSV;									//FB for saving binary file
	fbRecipeRename										:	FB_FileRename;
	bSetRecipeList										:	BOOL;										//Flag file not found -> create default	


	//Recipes list for table in user managment window
//	aRecipeIndexArray									:	ARRAY[0..udiMaxRecipeCount] OF DINT;		//Array of recipes (for table)
	aRecipeCaptionArray									:	ARRAY[0..3,0..udiMaxRecipeCount] OF WSTRING(120);	//Array of recipes (for table)
	diRecipeCaptionMaxIndex								:	DINT;										//Max index in aRecipeNameArray
	
	//Comon iterator for FOR/NEXT
	i													:	UDINT;										//iterator
	
	//Select item in user talble
	iSelectedArrayIndex									:	INT;										//Current selected recipe index in table
 	iPrevSelectedIndex									:	INT:=-1;									//Previous selected recipe for update
	wsSelectedCaption									:	WSTRING(120);
	iActualRecipeArrayIndex								:	INT :=-1;										//Current loaded recipe index in table
	bLineSelect											:	BOOL;										//Current selected recipe index in table
	udiSelectedRecipeIndex								:	UDINT;
	sProductBitmapId									:	STRING := 'C:\Recipe_photos\RecipeImages.1';
	
	//Region 'Window add new recipe'
	wsNewRecipeBase										:	WSTRING(80);
	bUseDefault											:	BOOL;
	
	udiNewRecipeIndex									:	UDINT;										//Window 'Add new recipe' : Recipe index
	wsNewRecipeCaption									:	WSTRING(80);								//Window 'Add new recipe' : 
	wsNewRecipeDescription								:	WSTRING(120);								//Window 'Add new recipe' : 
	bNewRecipeOk										:	BOOL;                                       //Window 'Add new recipe' : flag new recipe added
	bNewRecipeError										:	BOOL;                                       //Window 'Add new recipe' : flag new recipe adding error
	wsNewRecipeError									:	WSTRING;                                    //Window 'Add new recipe' : adding recipe error text description
	bAlreadyExist										:	BOOL;                                       //Window 'Add new recipe' : flag 'recipe with that name or index exist'

	
	iSaveRecipeCase										:	INT;
	iRenameRecipeCase									:	INT;
	iLoadRecipeCase										:	INT;
	diFileSaveIndex										:	DINT	:=-1;
	diFileLoadIndex										:	DINT	:=-1;
	
	bShowRecipeHomingWarning							:	BOOL;
	
	j													: 	UDINT;
	aSplit       : ARRAY[0..4] OF STRING(255);
    bResultSplit : BOOL;
	bTest:BOOL;	
	lrOldValue: LREAL;
	wsInfoCaption: WSTRING;
	
	bSort: BOOL;
	iColumnNumber: INT;
	diSelectedRecipeFileArrayIndex: DINT;
	
	stRecipe											:	ST_Recipe;
END_VAR

VAR_OUTPUT
END_VAR
VAR CONSTANT
	//WARNIG: uf you change this value you have to delet previous C:\RECIPES\LIST.BIN
	udiMaxRecipeCount									:	UDINT := 300;									//Max user count 
	udiMaxParamsVariablesCount							:	UDINT := 500;
END_VAR

VAR_IN_OUT
	
	//stRecipe											:	ST_Recipe;

END_VAR

ACT_Init();
ACT_UpdateList();
ACT_SaveRecipe();
ACT_LoadRecipe();
ACT_RenameRecipe();
IF bSort THEN
	METH_SortRecipesTable(0);
	bSort := FALSE;
END_IF

fbRecipeLoad();
fbRecipeSave(database 			:= 	ADR(aRecipeParamsValues));
fbRecipeRename();

fbListLoad();
fbListSave(database	 			:= 	ADR(aRecipeListString));

fbRecipeVariablesSave(database	:= 	ADR(aRecipeParamsVariables));
wsInfoNope:="";
//Tworzenie receptury
IF bCreateOrClone THEN
	Meth_CreateOrClone(FALSE);
END_IF

IF bNewRecipeOk THEN
	bCreateOrClone:=FALSE;
END_IF


//edycja nazwy
IF bRecipeShowEdit	 THEN
	METH_ShowEdit();
END_IF


IF bRecipeEdit		THEN
	METH_Edit();
END_IF

IF bEditOk THEN
	bRecipeEdit:=FALSE;
	bRecipeShowEdit:=FALSE;
END_IF
//Usuwanie receptury

IF bRecipeDelete THEN
	wsSelectedCaption:=aRecipeList[iSelectedArrayIndex].wsRecipeCaption;
	IF bRecipeDeleteAck THEN
		ACT_DeleteRecipe();
	END_IF
END_IF


//ładowanie receptury
IF bRecipeLoad THEN
	wsSelectedCaption:=aRecipeList[iSelectedArrayIndex].wsRecipeCaption;
	IF bRecipeLoadAck THEN
		IF (iLoadRecipeCase = 0) THEN
			iLoadRecipeCase	:=	10;
		END_IF
	END_IF
END_IF

IF bRecipeLoaded THEN
	bRecipeLoad:=FALSE;
	bRecipeLoadAck:=FALSE;
END_IF



//obróbka błędu

IF bEditFail THEN
	wsInfoNope:=wsEditErrorMessage;
ELSIF bNewRecipeError THEN
	wsInfoNope:=wsNewRecipeError;
END_IF

(*{warning 'Warning testy'}
stActRecipe.stP420_ExtInTransporter1.stTransporterVelocity.udiValue:=100;
stActRecipe.stP430_ExtInTransporter2.stTransporterVelocity.udiValue:=100;
stActRecipe.stP440_ExtInTransporter3dc.stTransporterVelocityL.udiValue:=100;
stActRecipe.stP440_ExtInTransporter3dc.stTransporterVelocityR.udiValue:=100;
stActRecipe.stP460_ExtInTransporter4dc.stTransporterVelocityL.udiValue:=100;
stActRecipe.stP460_ExtInTransporter4dc.stTransporterVelocityR.udiValue:=100;
stActRecipe.stP470_ExtInTransporter5.stTransporterVelocity.udiValue:=100;

stActRecipe.stP360_MacroTransportProcessRecipe.udiSensor430timeOff.udiValue	:= 1500;
stActRecipe.stP360_MacroTransportProcessRecipe.udiSensor430timeOn.udiValue	:= 1500;
stActRecipe.stP360_MacroTransportProcessRecipe.udiSensor440timeOff.udiValue	:= 1500;
stActRecipe.stP360_MacroTransportProcessRecipe.udiSensor440timeOn.udiValue	:= 1500;*)



(*tonCreateOrClone(IN:=(NOT bCreateOrClone), PT:=T#10S);

IF tonCreateOrClone.q THEN
	bAlreadyExist	:=	FALSE;
	bNewRecipeError	:=	FALSE;
	bNewRecipeOk	:=	FALSE;
END_IF*)

ACTION ACT_DeleteRecipe:
IF (iSelectedArrayIndex >=0) THEN
	IF (diSelectedRecipeFileArrayIndex>=0) THEN
		aRecipeList[diSelectedRecipeFileArrayIndex].bUsed:=FALSE;
		IF (udiUpdateCase = 0) THEN
			udiUpdateCase:=10;
		END_IF
	END_IF
END_IF
END_ACTION

ACTION ACT_Init:
CASE udiInitCase OF
	0:
//		fbListLoad.pStructAdr							:=	ADR(aRecipeList);
//		fbListLoad.udiStructSize						:=	SIZEOF(aRecipeList);
		fbListLoad.sFilePath							:=	'C:\Recipes\List.CSV';
		fbListLoad.database								:= 	ADR(aRecipeListString);
		fbListLoad.nRows								:= 	udiMaxRecipeCount;
		fbListLoad.nCols								:= 	0;		
		
//		fbListSave.pStructAdr							:=	ADR(aRecipeList);
//		fbListSave.udiStructSize						:=	SIZEOF(aRecipeList);
//		fbListSave.database								:= 	ADR(aRecipeListString);
		fbListSave.nRows								:= 	udiMaxRecipeCount;
		fbListSave.nCols								:= 	0;
		
		fbListSave.sFilePath							:=	'C:\Recipes\List.CSV';
			
//		fbRecipeLoad.pStructAdr							:=  ADR(stFileRecipe);
//		fbRecipeLoad.udiStructSize						:=  SIZEOF(stFileRecipe);
		
		fbRecipeVariablesSave.sFilePath					:=	'C:\Recipes\ParamVariables.CSV';		
//		fbRecipeVariablesSave.database					:= 	ADR(aRecipeParamsVariables);
		fbRecipeVariablesSave.nRows						:= 	udiMaxParamsVariablesCount;
		fbRecipeVariablesSave.nCols						:= 	0;
		
		udiInitCase										:=	10;
	
	10:
		fbListLoad.bExecute								:=	TRUE;
		udiInitCase										:=	20;
	20:
		IF (fbListLoad.bDone) THEN
			fbListLoad.bExecute							:=	FALSE;
			udiInitCase									:=	60;
		END_IF
		IF (fbListLoad.bError) THEN
			fbListLoad.bExecute							:=	FALSE;
			udiInitCase									:=	10;
		END_IF
//	30:
//		udiInitCase										:=	40;
//	
//	40:
//		fbListSave.bExecute								:=	TRUE;
//		udiInitCase										:=	50;
//	50:
//		IF (fbListSave.bDone) THEN
//			fbListSave.bExecute							:=	FALSE;
//			udiInitCase									:=	60;
//		END_IF
//		IF (fbListSave.bError) THEN
//			fbListSave.bExecute							:=	FALSE;
//			udiInitCase									:=	60;
//		END_IF
	60:
			METH_RecipeFileInit();	
			fbRecipeVariablesSave.bExecute				:=	TRUE;
			udiInitCase									:=	70;	
	70:
		IF (fbRecipeVariablesSave.bDone) THEN
			fbRecipeVariablesSave.bExecute				:=	FALSE;
			udiInitCase									:=	100;
		END_IF
		IF (fbRecipeVariablesSave.bError) THEN
			fbRecipeVariablesSave.bExecute				:=	FALSE;
			udiInitCase									:=	100;
		END_IF			
	100:
		METH_ParseRecipesListStringArray();
		METH_CreateRecipesListStringArray();	
		diRecipeCaptionMaxIndex									:=	-1;
		FOR i:=0 TO udiMaxRecipeCount DO
			IF (aRecipeList[i].bUsed) THEN
				diRecipeCaptionMaxIndex							:=	diRecipeCaptionMaxIndex +1;
//				aRecipeIndexArray[diRecipeCaptionMaxIndex]		:=	UDINT_TO_DINT(i);
				aRecipeCaptionArray[0,diRecipeCaptionMaxIndex]	:=	UDINT_TO_WSTRING(aRecipeList[i].udiIndex);
				aRecipeCaptionArray[1,diRecipeCaptionMaxIndex]	:=	aRecipeList[i].wsRecipeCaption;
				aRecipeCaptionArray[2,diRecipeCaptionMaxIndex]	:=	aRecipeList[i].wsCreateDate;				
			END_IF
		END_FOR
		


IF (NOT bInit) THEN
	stRecipe.stUBL.bBadBottleConveyorEnableShow.bDefault:=FALSE;
	stRecipe.stUBL.bPucksInserterEnableShow.bDefault:=TRUE;
	stRecipe.stUBL.bROPPCappingEnableShow.bDefault:=FALSE;
	stRecipe.stUBL.bROPPDragEnableShow.bDefault:=TRUE;
	stRecipe.stUBL.bROPPFeederEnableShow.bDefault:=FALSE;
	stRecipe.stUBL.bROPPSlowerEnableShow.bDefault:=TRUE;
	stRecipe.stUBL.bBadBottleConveyorEnableShow.bDefault:=TRUE;
	stRecipe.stUBL.bBottleDragingStationEnableShow.bDefault:=TRUE;
	stRecipe.stUBL.bBottleFeederEnableShow.bDefault:=FALSE;
	stRecipe.stUBL.bBottleTransferEnableShow.bDefault:=TRUE;
	stRecipe.stUBL.bBottleTransferInkJetEnableShow.bDefault:=TRUE;
	stRecipe.stUBL.bBottleTransferPickOnlyOneShow.bDefault:=FALSE;
	stRecipe.stUBL.bBottleTransferWeightEnableShow.bDefault:=FALSE;
	stRecipe.stUBL.bCapCorrectCheckCameraEnableShow.bDefault:=FALSE;
	stRecipe.stUBL.bCapCorrectCheckEnableShow.bDefault:=TRUE;
    stRecipe.stUBL.bCapFeederEnableShow.bDefault:=FALSE;
    stRecipe.stUBL.bCapFeederGateEnableShow.bDefault:=FALSE;
    stRecipe.stUBL.bCapPuttedCheckEnableShow.bDefault:=TRUE;
    stRecipe.stUBL.bCapSorterDragEnableShow.bDefault:=TRUE;
    stRecipe.stUBL.bCapSorterOnlyWeightOKEnableShow.bDefault:=FALSE;
    stRecipe.stUBL.bCircularInkjetEnableShow.bDefault:=FALSE;
    stRecipe.stUBL.bDispencer1DoseSuckingShow.bDefault:=FALSE;
    stRecipe.stUBL.bDispencer1EnableShow.bDefault:=TRUE;
    stRecipe.stUBL.bDispencer1LiftSynchroPh1Show.bDefault:=FALSE;
    stRecipe.stUBL.bDispencer1LiftSynchroPh2Show.bDefault:=TRUE;
    stRecipe.stUBL.bDispencer1LiftSynchroPh3Show.bDefault:=TRUE;
    stRecipe.stUBL.bDispencer1WeightCorrectionEnableShow.bDefault:=TRUE;
    stRecipe.stUBL.bDispencer2DoseSuckingShow.bDefault:=FALSE;
    stRecipe.stUBL.bDispencer2EnableShow.bDefault:=TRUE;
    stRecipe.stUBL.bDispencer2LiftSynchroPh1Show.bDefault:=FALSE;
    stRecipe.stUBL.bDispencer2LiftSynchroPh2Show.bDefault:=TRUE;
    stRecipe.stUBL.bDispencer2LiftSynchroPh3Show.bDefault:=TRUE;
    stRecipe.stUBL.bDispencer2WeightCorrectionEnableShow.bDefault:=TRUE;
    stRecipe.stUBL.bDispencer3EnableShow.bDefault:=TRUE;
    stRecipe.stUBL.bDispencer3WeightCorrectionEnableShow.bDefault:=TRUE;
    stRecipe.stUBL.bDispencer4EnableShow.bDefault:=TRUE;
    stRecipe.stUBL.bDispencer4WeightCorrectionEnableShow.bDefault:=TRUE;
    stRecipe.stUBL.bDispencersCatchEnableShow.bDefault:=TRUE;
    stRecipe.stUBL.bDispencersCatchMaxPressureShow.bDefault:=TRUE;
    stRecipe.stUBL.bDosingTwoPhasesShow.bDefault:=FALSE;
    stRecipe.stUBL.bExEnableShow.bDefault:=FALSE;
	stRecipe.stUBL.bExitTurnTable1EnableShow.bDefault:=FALSE;
	stRecipe.stUBL.bFormTransportersEnableShow.bDefault:=TRUE;
	stRecipe.stUBL.bFormsDragingLeftEnableShow.bDefault:=TRUE;
	stRecipe.stUBL.bFormsDragingRightEnableShow.bDefault:=TRUE;
	stRecipe.stUBL.bGateAfterWeightEnableShow.bDefault:=TRUE;
	stRecipe.stUBL.bGateBeforeDispencersEnableShow.bDefault:=TRUE;
	stRecipe.stUBL.bGateRobotEnableShow.bDefault:=TRUE;
	stRecipe.stUBL.bGripperScrewer1EnableShow.bDefault:=TRUE;
	stRecipe.stUBL.bGripperScrewer1FindScrewShow.bDefault:=TRUE;
	stRecipe.stUBL.bGripperScrewer1Option1Show.bDefault:=FALSE;
	stRecipe.stUBL.bGripperScrewer1Option2Show.bDefault:=FALSE;
	stRecipe.stUBL.bGripperScrewer1Option3Show.bDefault:=TRUE;
	stRecipe.stUBL.bGripperScrewer1Option4Show.bDefault:=FALSE;
	stRecipe.stUBL.bGripperScrewer1Option5Show.bDefault:=FALSE;
	stRecipe.stUBL.bGripperScrewer1Option6Show.bDefault:=FALSE;
	stRecipe.stUBL.bGripperScrewer1Option7Show.bDefault:=TRUE;
	stRecipe.stUBL.bGripperScrewer2EnableShow.bDefault:=TRUE;
	stRecipe.stUBL.bLabelMachineEnableShow.bDefault:=FALSE;
	stRecipe.stUBL.bLidFeederDragingStationEnableShow.bDefault:=FALSE;
	stRecipe.stUBL.bLidFeederEnableShow.bDefault:=FALSE;
	stRecipe.stUBL.bLidFeederHeaterEnableShow.bDefault:=FALSE;
	stRecipe.stUBL.bLidPuttedCheckEnableShow.bDefault:=FALSE;
	stRecipe.stUBL.bLidSealerDragingStationEnableShow.bDefault:=FALSE;
	stRecipe.stUBL.bLidSealerEnableShow.bDefault:=FALSE;
	stRecipe.stUBL.bLidSealerHeaterEnableShow.bDefault:=FALSE;
	stRecipe.stUBL.bTank1LevelSignalInvertShow.bDefault:=FALSE;
	stRecipe.stUBL.bTank1MixerEnableShow.bDefault:=FALSE;
	stRecipe.stUBL.bTank1PressureEnableShow.bDefault:=FALSE;
	stRecipe.stUBL.bTank1SupplyPumpEnableShow.bDefault:=FALSE;
	stRecipe.stUBL.bTank2LevelSignalInvertShow.bDefault:=FALSE;
	stRecipe.stUBL.bTank2SupplyPumpEnableShow.bDefault:=FALSE;
	stRecipe.stUBL.bTankHeatingEnableShow.bDefault:=FALSE;
	stRecipe.stUBL.bWeight1EnableShow.bDefault:=TRUE;
	
	stRecipe.stUBL.iPucksInserterAllowFormDelayShow.diDefault:=5000;
	stRecipe.stUBL.iPucksInserterAllowFormDelayShow.diMinLimit:=0;
	stRecipe.stUBL.iPucksInserterAllowFormDelayShow.diMaxLimit:=10000;	
	
	stRecipe.stUBL.iPucksInserterBottleSensorDelayShow.diDefault:=100;
	stRecipe.stUBL.iPucksInserterBottleSensorDelayShow.diMinLimit:=0;
	stRecipe.stUBL.iPucksInserterBottleSensorDelayShow.diMaxLimit:=1000;
	
	stRecipe.stUBL.iPucksInserterConveyorVelocitySVShow.udiDefault:=900;
	stRecipe.stUBL.iPucksInserterConveyorVelocitySVShow.udiMinLimit:=100;
	stRecipe.stUBL.iPucksInserterConveyorVelocitySVShow.udiMaxLimit:=1200;
	
	stRecipe.stUBL.iPucksInserterFormGateDelayShow.diDefault:=200;
	stRecipe.stUBL.iPucksInserterFormGateDelayShow.diMinLimit:=0;
	stRecipe.stUBL.iPucksInserterFormGateDelayShow.diMaxLimit:=1000;
	
	stRecipe.stUBL.iPucksInserterTurntableVelocitySVShow.udiDefault:=900;
	stRecipe.stUBL.iPucksInserterTurntableVelocitySVShow.udiMinLimit:=100;
	stRecipe.stUBL.iPucksInserterTurntableVelocitySVShow.udiMaxLimit:=1200;
	
	stRecipe.stUBL.lrPucksInserterHammerHeightSVShow.lrDefault:=285;
	stRecipe.stUBL.lrPucksInserterHammerHeightSVShow.lrMinLimit:=0;
	stRecipe.stUBL.lrPucksInserterHammerHeightSVShow.lrMaxLimit:=2100;
	
	stRecipe.stUBL.lrPucksInserterWheelAccelerationShow.lrDefault:=2000;
	stRecipe.stUBL.lrPucksInserterWheelAccelerationShow.lrMinLimit:=0;
	stRecipe.stUBL.lrPucksInserterWheelAccelerationShow.lrMaxLimit:=2100;
	
	stRecipe.stUBL.lrPucksInserterWheelOffsetShow.lrDefault:=3;
	stRecipe.stUBL.lrPucksInserterWheelOffsetShow.lrMinLimit:=-10;
	stRecipe.stUBL.lrPucksInserterWheelOffsetShow.lrMaxLimit:=10;

	stRecipe.stUBL.lrPucksInserterWheelVelocityShow.lrDefault:=1600;
	stRecipe.stUBL.lrPucksInserterWheelVelocityShow.lrMinLimit:=0;
	stRecipe.stUBL.lrPucksInserterWheelVelocityShow.lrMaxLimit:=2100;

	stRecipe.stUBL.nExitConveyorVelocitySVShow.udiDefault:=1200;
	stRecipe.stUBL.nExitConveyorVelocitySVShow.udiMinLimit:=0;
	stRecipe.stUBL.nExitConveyorVelocitySVShow.udiMaxLimit:=1500;

	stRecipe.stUBL.iROPPCapping1ToolShow.diDefault:=1;
	stRecipe.stUBL.iROPPCapping1ToolShow.diMinLimit:=1;
	stRecipe.stUBL.iROPPCapping1ToolShow.diMaxLimit:=2;

	stRecipe.stUBL.iROPPCappingTime2Show.diDefault:=200;
	stRecipe.stUBL.iROPPCappingTime2Show.diMinLimit:=0;
	stRecipe.stUBL.iROPPCappingTime2Show.diMaxLimit:=350;

	stRecipe.stUBL.iROPPCappingTimeShow.diDefault:=200;
	stRecipe.stUBL.iROPPCappingTimeShow.diMinLimit:=0;
	stRecipe.stUBL.iROPPCappingTimeShow.diMaxLimit:=350;

	stRecipe.stUBL.iROPPFeederTimeDelayOffShow.diDefault:=300;
	stRecipe.stUBL.iROPPFeederTimeDelayOffShow.diMinLimit:=0;
	stRecipe.stUBL.iROPPFeederTimeDelayOffShow.diMaxLimit:=1000;

	stRecipe.stUBL.iROPPFeederTimeDelayOnShow.diDefault:=300;
	stRecipe.stUBL.iROPPFeederTimeDelayOnShow.diMinLimit:=0;
	stRecipe.stUBL.iROPPFeederTimeDelayOnShow.diMaxLimit:=350;

	stRecipe.stUBL.iROPPFeederTimeToEmptySleeveErrorShow.diDefault:=120;
	stRecipe.stUBL.iROPPFeederTimeToEmptySleeveErrorShow.diMinLimit:=10;
	stRecipe.stUBL.iROPPFeederTimeToEmptySleeveErrorShow.diMaxLimit:=120;

	stRecipe.stUBL.lrROPPCappingHeightPosSVShow.lrDefault:=195;
	stRecipe.stUBL.lrROPPCappingHeightPosSVShow.lrMinLimit:=0;
	stRecipe.stUBL.lrROPPCappingHeightPosSVShow.lrMaxLimit:=1000;

	stRecipe.stUBL.lrROPPCappingVelocitySVShow.lrDefault:=800;
	stRecipe.stUBL.lrROPPCappingVelocitySVShow.lrMinLimit:=0;
	stRecipe.stUBL.lrROPPCappingVelocitySVShow.lrMaxLimit:=1000;

	stRecipe.stUBL.lrROPPDragAccelerationShow.lrDefault:=2400;
	stRecipe.stUBL.lrROPPDragAccelerationShow.lrMinLimit:=100;
	stRecipe.stUBL.lrROPPDragAccelerationShow.lrMaxLimit:=10000;

	stRecipe.stUBL.lrROPPDragDecelerationShow.lrDefault:=2400;
	stRecipe.stUBL.lrROPPDragDecelerationShow.lrMinLimit:=100;
	stRecipe.stUBL.lrROPPDragDecelerationShow.lrMaxLimit:=10000;

	stRecipe.stUBL.lrROPPDragVelocityShow.lrDefault:=380;
	stRecipe.stUBL.lrROPPDragVelocityShow.lrMinLimit:=100;
	stRecipe.stUBL.lrROPPDragVelocityShow.lrMaxLimit:=10000;

	stRecipe.stUBL.lrROPPFeederHeightPosSVShow.lrDefault:=200;
	stRecipe.stUBL.lrROPPFeederHeightPosSVShow.lrMinLimit:=0;
	stRecipe.stUBL.lrROPPFeederHeightPosSVShow.lrMaxLimit:=350;

	stRecipe.stUBL.nROPPSlowerVelocitySVShow.udiDefault:=1800;
	stRecipe.stUBL.nROPPSlowerVelocitySVShow.udiMinLimit:=100;
	stRecipe.stUBL.nROPPSlowerVelocitySVShow.udiMaxLimit:=2100;

	stRecipe.stUBL.iBottleFeederAllowFormDelayShow.diDefault:=5000;
	stRecipe.stUBL.iBottleFeederAllowFormDelayShow.diMinLimit:=0;
	stRecipe.stUBL.iBottleFeederAllowFormDelayShow.diMaxLimit:=10000;
	
	stRecipe.stUBL.iBottleFeederBottleSensorDelayShow.diDefault:=100;
	stRecipe.stUBL.iBottleFeederBottleSensorDelayShow.diMinLimit:=0;
	stRecipe.stUBL.iBottleFeederBottleSensorDelayShow.diMaxLimit:=1000;
	
	stRecipe.stUBL.iBottleFeederFormGateDelayShow.diDefault:=200;
	stRecipe.stUBL.iBottleFeederFormGateDelayShow.diMinLimit:=0;
	stRecipe.stUBL.iBottleFeederFormGateDelayShow.diMaxLimit:=1000;
	
	stRecipe.stUBL.iBottleFeederTurntableVelocitySVShow.udiDefault:=900;
	stRecipe.stUBL.iBottleFeederTurntableVelocitySVShow.udiMinLimit:=100;
	stRecipe.stUBL.iBottleFeederTurntableVelocitySVShow.udiMaxLimit:=2100;
	
	stRecipe.stUBL.iBottleTransferPick2OffsetXShow.diDefault:=0;
	stRecipe.stUBL.iBottleTransferPick2OffsetXShow.diMinLimit:=-1000;
	stRecipe.stUBL.iBottleTransferPick2OffsetXShow.diMaxLimit:=1000;

	stRecipe.stUBL.iBottleTransferPick2OffsetYShow.diDefault:=0;
	stRecipe.stUBL.iBottleTransferPick2OffsetYShow.diMinLimit:=-1000;
	stRecipe.stUBL.iBottleTransferPick2OffsetYShow.diMaxLimit:=1000;
	
	stRecipe.stUBL.iBottleTransferPick2OffsetZShow.diDefault:=0;
	stRecipe.stUBL.iBottleTransferPick2OffsetZShow.diMinLimit:=-1000;
	stRecipe.stUBL.iBottleTransferPick2OffsetZShow.diMaxLimit:=1000;

	stRecipe.stUBL.iBottleTransferPickOffsetXShow.diDefault:=0;
	stRecipe.stUBL.iBottleTransferPickOffsetXShow.diMinLimit:=-1000;
	stRecipe.stUBL.iBottleTransferPickOffsetXShow.diMaxLimit:=1000;

	stRecipe.stUBL.iBottleTransferPickOffsetYShow.diDefault:=0;
	stRecipe.stUBL.iBottleTransferPickOffsetYShow.diMinLimit:=-1000;
	stRecipe.stUBL.iBottleTransferPickOffsetYShow.diMaxLimit:=1000;

	stRecipe.stUBL.iBottleTransferPickOffsetZShow.diDefault:=0;
	stRecipe.stUBL.iBottleTransferPickOffsetZShow.diMinLimit:=-1000;
	stRecipe.stUBL.iBottleTransferPickOffsetZShow.diMaxLimit:=1000;

	stRecipe.stUBL.iBottleTransferPlace1OffsetXShow.diDefault:=0;
	stRecipe.stUBL.iBottleTransferPlace1OffsetXShow.diMinLimit:=-1000;
	stRecipe.stUBL.iBottleTransferPlace1OffsetXShow.diMaxLimit:=1000;

	stRecipe.stUBL.iBottleTransferPlace1OffsetYShow.diDefault:=0;
	stRecipe.stUBL.iBottleTransferPlace1OffsetYShow.diMinLimit:=-1000;
	stRecipe.stUBL.iBottleTransferPlace1OffsetYShow.diMaxLimit:=1000;

	stRecipe.stUBL.iBottleTransferPlace1OffsetZShow.diDefault:=0;
	stRecipe.stUBL.iBottleTransferPlace1OffsetZShow.diMinLimit:=-1000;
	stRecipe.stUBL.iBottleTransferPlace1OffsetZShow.diMaxLimit:=1000;

	stRecipe.stUBL.iBottleTransferPlace2OffsetXShow.diDefault:=0;
	stRecipe.stUBL.iBottleTransferPlace2OffsetXShow.diMinLimit:=-1000;
	stRecipe.stUBL.iBottleTransferPlace2OffsetXShow.diMaxLimit:=1000;

	stRecipe.stUBL.iBottleTransferPlace2OffsetYShow.diDefault:=0;
	stRecipe.stUBL.iBottleTransferPlace2OffsetYShow.diMinLimit:=-1000;
	stRecipe.stUBL.iBottleTransferPlace2OffsetYShow.diMaxLimit:=1000;

	stRecipe.stUBL.iBottleTransferPlace2OffsetZShow.diDefault:=0;
	stRecipe.stUBL.iBottleTransferPlace2OffsetZShow.diMinLimit:=-1000;
	stRecipe.stUBL.iBottleTransferPlace2OffsetZShow.diMaxLimit:=1000;

	stRecipe.stUBL.iBottleTransferSpeedShow.diDefault:=20;
	stRecipe.stUBL.iBottleTransferSpeedShow.diMinLimit:=0;
	stRecipe.stUBL.iBottleTransferSpeedShow.diMaxLimit:=100;

	stRecipe.stUBL.iBottleTransferWeightIntervalShow.diDefault:=0;
	stRecipe.stUBL.iBottleTransferWeightIntervalShow.diMinLimit:=0;
	stRecipe.stUBL.iBottleTransferWeightIntervalShow.diMaxLimit:=1000;

	stRecipe.stUBL.iCapCorrectCheckCameraProgramShow.diDefault:=0;
	stRecipe.stUBL.iCapCorrectCheckCameraProgramShow.diMinLimit:=0;
	stRecipe.stUBL.iCapCorrectCheckCameraProgramShow.diMaxLimit:=1000;

	stRecipe.stUBL.iCapFeederTimeDelayOffShow.diDefault:=100;
	stRecipe.stUBL.iCapFeederTimeDelayOffShow.diMinLimit:=0;
    stRecipe.stUBL.iCapFeederTimeDelayOffShow.diMaxLimit:=5000;

	stRecipe.stUBL.iCapFeederTimeDelayOnShow.diDefault:=1000;
	stRecipe.stUBL.iCapFeederTimeDelayOnShow.diMinLimit:=0;
	stRecipe.stUBL.iCapFeederTimeDelayOnShow.diMaxLimit:=5000;

	stRecipe.stUBL.iCapFeederTimeToEmptySleeveErrorShow.diDefault:=30;
	stRecipe.stUBL.iCapFeederTimeToEmptySleeveErrorShow.diMinLimit:=10;
    stRecipe.stUBL.iCapFeederTimeToEmptySleeveErrorShow.diMaxLimit:=120;

	stRecipe.stUBL.iGripperScrewer1StartDelayShow.diDefault:=0;
	stRecipe.stUBL.iGripperScrewer1StartDelayShow.diMinLimit:=0;
	stRecipe.stUBL.iGripperScrewer1StartDelayShow.diMaxLimit:=10000;

	stRecipe.stUBL.iGripperScrewer1ToolShow.diDefault:=0;
	stRecipe.stUBL.iGripperScrewer1ToolShow.diMinLimit:=0;
	stRecipe.stUBL.iGripperScrewer1ToolShow.diMaxLimit:=10;

	stRecipe.stUBL.iLidFeeder1TempSVShow.diDefault:=100;
	stRecipe.stUBL.iLidFeeder1TempSVShow.diMinLimit:=0;
	stRecipe.stUBL.iLidFeeder1TempSVShow.diMaxLimit:=350;

	stRecipe.stUBL.iLidFeeder2TempSVShow.diDefault:=100;
	stRecipe.stUBL.iLidFeeder2TempSVShow.diMinLimit:=0;
	stRecipe.stUBL.iLidFeeder2TempSVShow.diMaxLimit:=350;

	stRecipe.stUBL.iLidFeederHeatingTimeShow.diDefault:=200;
	stRecipe.stUBL.iLidFeederHeatingTimeShow.diMinLimit:=0;
	stRecipe.stUBL.iLidFeederHeatingTimeShow.diMaxLimit:=1000;

	stRecipe.stUBL.iLidFeederTempHisteresisShow.diDefault:=10;
	stRecipe.stUBL.iLidFeederTempHisteresisShow.diMinLimit:=0;
	stRecipe.stUBL.iLidFeederTempHisteresisShow.diMaxLimit:=350;

	stRecipe.stUBL.iLidSealer1TempSVShow.diDefault:=100;
	stRecipe.stUBL.iLidSealer1TempSVShow.diMinLimit:=0;
	stRecipe.stUBL.iLidSealer1TempSVShow.diMaxLimit:=350;

	stRecipe.stUBL.iLidSealer2TempSVShow.diDefault:=100;
	stRecipe.stUBL.iLidSealer2TempSVShow.diMinLimit:=0;
	stRecipe.stUBL.iLidSealer2TempSVShow.diMaxLimit:=350;

	stRecipe.stUBL.iLidSealerHeatingTimeShow.diDefault:=200;
    stRecipe.stUBL.iLidSealerHeatingTimeShow.diMinLimit:=0;
	stRecipe.stUBL.iLidSealerHeatingTimeShow.diMaxLimit:=1000;

	stRecipe.stUBL.iLidSealerTempHisteresisShow.diDefault:=10;
    stRecipe.stUBL.iLidSealerTempHisteresisShow.diMinLimit:=0;
	stRecipe.stUBL.iLidSealerTempHisteresisShow.diMaxLimit:=350;

	stRecipe.stUBL.iTankHeatingTempSVShow.diDefault:=60;
	stRecipe.stUBL.iTankHeatingTempSVShow.diMinLimit:=0;
	stRecipe.stUBL.iTankHeatingTempSVShow.diMaxLimit:=100;
	
    stRecipe.stUBL.iWeightCorrectionNumberOfSamplesShow.udiDefault:=2;
	stRecipe.stUBL.iWeightCorrectionNumberOfSamplesShow.udiMinLimit:=0;
	stRecipe.stUBL.iWeightCorrectionNumberOfSamplesShow.udiMaxLimit:=100;
	
    stRecipe.stUBL.lrBottleDragingStationVelocityShow.lrDefault:=380;
	stRecipe.stUBL.lrBottleDragingStationVelocityShow.lrMinLimit:=0;
	stRecipe.stUBL.lrBottleDragingStationVelocityShow.lrMaxLimit:=1000;
	
    stRecipe.stUBL.lrCapCorrectCheckHeightPosSVShow.lrDefault:=200.5;
	stRecipe.stUBL.lrCapCorrectCheckHeightPosSVShow.lrMinLimit:=0;
	stRecipe.stUBL.lrCapCorrectCheckHeightPosSVShow.lrMaxLimit:=1000;
	
    stRecipe.stUBL.lrCapFeederHeightPosSVShow.lrDefault:=205.4;
	stRecipe.stUBL.lrCapFeederHeightPosSVShow.lrMinLimit:=50;
	stRecipe.stUBL.lrCapFeederHeightPosSVShow.lrMaxLimit:=350;
	
    stRecipe.stUBL.lrCapPuttedCheckHeightPosSVShow.lrDefault:=203;
	stRecipe.stUBL.lrCapPuttedCheckHeightPosSVShow.lrMinLimit:=-10000;
	stRecipe.stUBL.lrCapPuttedCheckHeightPosSVShow.lrMaxLimit:=10000;
	
    stRecipe.stUBL.lrCapSorterDragAccelerationShow.lrDefault:=2400;
	stRecipe.stUBL.lrCapSorterDragAccelerationShow.lrMinLimit:=1;
	stRecipe.stUBL.lrCapSorterDragAccelerationShow.lrMaxLimit:=5000;
	
    stRecipe.stUBL.lrCapSorterDragDecelerationShow.lrDefault:=2400;
	stRecipe.stUBL.lrCapSorterDragDecelerationShow.lrMinLimit:=1;
	stRecipe.stUBL.lrCapSorterDragDecelerationShow.lrMaxLimit:=5000;
	
    stRecipe.stUBL.lrCapSorterDragVelocityShow.lrDefault:=380;
	stRecipe.stUBL.lrCapSorterDragVelocityShow.lrMinLimit:=1;
	stRecipe.stUBL.lrCapSorterDragVelocityShow.lrMaxLimit:=1000;
	
    stRecipe.stUBL.lrCupWeightShow.lrDefault:=0;
	stRecipe.stUBL.lrCupWeightShow.lrMinLimit:=0;
	stRecipe.stUBL.lrCupWeightShow.lrMaxLimit:=1000;
	
    stRecipe.stUBL.lrDispencer1DoseSuckingTimeDelayShow.lrDefault:=0;
	stRecipe.stUBL.lrDispencer1DoseSuckingTimeDelayShow.lrMinLimit:=0;
	stRecipe.stUBL.lrDispencer1DoseSuckingTimeDelayShow.lrMaxLimit:=1000;
	
    stRecipe.stUBL.lrDispencer1DoseSuckingVolumeShow.lrDefault:=0;
	stRecipe.stUBL.lrDispencer1DoseSuckingVolumeShow.lrMinLimit:=0;
	stRecipe.stUBL.lrDispencer1DoseSuckingVolumeShow.lrMaxLimit:=1000;
	
    stRecipe.stUBL.lrDispencer1DoseValveCloseTimeDecShow.lrDefault:=0;
	stRecipe.stUBL.lrDispencer1DoseValveCloseTimeDecShow.lrMinLimit:=0;
	stRecipe.stUBL.lrDispencer1DoseValveCloseTimeDecShow.lrMaxLimit:=1000;
	
    stRecipe.stUBL.lrDispencer1DoseValveCloseVolumeShow.lrDefault:=1;
	stRecipe.stUBL.lrDispencer1DoseValveCloseVolumeShow.lrMinLimit:=0;
	stRecipe.stUBL.lrDispencer1DoseValveCloseVolumeShow.lrMaxLimit:=1000;
	
	stRecipe.stUBL.udiDispencer1DosingDoneDelayTimeShow.udiDefault:=0;
	stRecipe.stUBL.udiDispencer1DosingDoneDelayTimeShow.udiMinLimit:=0;
	stRecipe.stUBL.udiDispencer1DosingDoneDelayTimeShow.udiMaxLimit:=1000;
	
    stRecipe.stUBL.lrDispencer1DoseValveOpenTimeAccShow.lrDefault:=200;
	stRecipe.stUBL.lrDispencer1DoseValveOpenTimeAccShow.lrMinLimit:=0;
	stRecipe.stUBL.lrDispencer1DoseValveOpenTimeAccShow.lrMaxLimit:=1000;
	
    stRecipe.stUBL.lrDispencer1DoseVolumeShow.lrDefault:=495;
	stRecipe.stUBL.lrDispencer1DoseVolumeShow.lrMinLimit:=0;
	stRecipe.stUBL.lrDispencer1DoseVolumeShow.lrMaxLimit:=1000;	
	
    stRecipe.stUBL.lrDispencer1LifterStartDosePositionShow.lrDefault:=80;
	stRecipe.stUBL.lrDispencer1LifterStartDosePositionShow.lrMinLimit:=-1000;
	stRecipe.stUBL.lrDispencer1LifterStartDosePositionShow.lrMaxLimit:=1000;
	
	stRecipe.stUBL.uiDispencerStartDosingDelayShow.udiDefault:=0;
	stRecipe.stUBL.uiDispencerStartDosingDelayShow.udiMinLimit:=0;
	stRecipe.stUBL.uiDispencerStartDosingDelayShow.udiMaxLimit:=10000;
	
    stRecipe.stUBL.lrDispencer1LifterStopDosePositionShow.lrDefault:=192;
	stRecipe.stUBL.lrDispencer1LifterStopDosePositionShow.lrMinLimit:=-1000;
	stRecipe.stUBL.lrDispencer1LifterStopDosePositionShow.lrMaxLimit:=1000;    
	
    stRecipe.stUBL.lrDispencer1Phase1AccelerationShow.lrDefault:=600;
	stRecipe.stUBL.lrDispencer1Phase1AccelerationShow.lrMinLimit:=1;
	stRecipe.stUBL.lrDispencer1Phase1AccelerationShow.lrMaxLimit:=100000;
	
    stRecipe.stUBL.lrDispencer1Phase1DecelerationShow.lrDefault:=150;
	stRecipe.stUBL.lrDispencer1Phase1DecelerationShow.lrMinLimit:=1;
	stRecipe.stUBL.lrDispencer1Phase1DecelerationShow.lrMaxLimit:=100000;
	
    stRecipe.stUBL.lrDispencer1Phase1VelocityShow.lrDefault:=140;
	stRecipe.stUBL.lrDispencer1Phase1VelocityShow.lrMinLimit:=1;
	stRecipe.stUBL.lrDispencer1Phase1VelocityShow.lrMaxLimit:=10000;
	
    stRecipe.stUBL.lrDispencer1Phase1VolumeShow.lrDefault:=0;
	stRecipe.stUBL.lrDispencer1Phase1VolumeShow.lrMinLimit:=0;
	stRecipe.stUBL.lrDispencer1Phase1VolumeShow.lrMaxLimit:=1000;
	
    stRecipe.stUBL.lrDispencer1Phase2AccelerationShow.lrDefault:=400;
	stRecipe.stUBL.lrDispencer1Phase2AccelerationShow.lrMinLimit:=1;
	stRecipe.stUBL.lrDispencer1Phase2AccelerationShow.lrMaxLimit:=100000;
	
    stRecipe.stUBL.lrDispencer1Phase2DecelerationShow.lrDefault:=2000;
	stRecipe.stUBL.lrDispencer1Phase2DecelerationShow.lrMinLimit:=1;
	stRecipe.stUBL.lrDispencer1Phase2DecelerationShow.lrMaxLimit:=100000;	
	
    stRecipe.stUBL.lrDispencer1Phase2VelocityShow.lrDefault:=140;
	stRecipe.stUBL.lrDispencer1Phase2VelocityShow.lrMinLimit:=1;
	stRecipe.stUBL.lrDispencer1Phase2VelocityShow.lrMaxLimit:=10000;
	
    stRecipe.stUBL.lrDispencer1Phase2VolumeShow.lrDefault:=0;
	stRecipe.stUBL.lrDispencer1Phase2VolumeShow.lrMinLimit:=0;
	stRecipe.stUBL.lrDispencer1Phase2VolumeShow.lrMaxLimit:=1000;
	
    stRecipe.stUBL.lrDispencer1Phase3AccelerationShow.lrDefault:=50;
	stRecipe.stUBL.lrDispencer1Phase3AccelerationShow.lrMinLimit:=1;
	stRecipe.stUBL.lrDispencer1Phase3AccelerationShow.lrMaxLimit:=100000;
	
    stRecipe.stUBL.lrDispencer1Phase3DecelerationShow.lrDefault:=50;
	stRecipe.stUBL.lrDispencer1Phase3DecelerationShow.lrMinLimit:=1;
	stRecipe.stUBL.lrDispencer1Phase3DecelerationShow.lrMaxLimit:=100000;
	
    stRecipe.stUBL.lrDispencer1Phase3VelocityShow.lrDefault:=50;
	stRecipe.stUBL.lrDispencer1Phase3VelocityShow.lrMinLimit:=1;
	stRecipe.stUBL.lrDispencer1Phase3VelocityShow.lrMaxLimit:=10000;
	
    stRecipe.stUBL.lrDispencer1SuckAccelerationShow.lrDefault:=3000;
	stRecipe.stUBL.lrDispencer1SuckAccelerationShow.lrMinLimit:=1;
	stRecipe.stUBL.lrDispencer1SuckAccelerationShow.lrMaxLimit:=100000;
	
    stRecipe.stUBL.lrDispencer1SuckValveCloseTimeDelayShow.lrDefault:=0;
	stRecipe.stUBL.lrDispencer1SuckValveCloseTimeDelayShow.lrMinLimit:=0;
	stRecipe.stUBL.lrDispencer1SuckValveCloseTimeDelayShow.lrMaxLimit:=4000;
	
    stRecipe.stUBL.lrDispencer1SuckValveOpenTimeDelayShow.lrDefault:=0;
	stRecipe.stUBL.lrDispencer1SuckValveOpenTimeDelayShow.lrMinLimit:=0;
	stRecipe.stUBL.lrDispencer1SuckValveOpenTimeDelayShow.lrMaxLimit:=1000;
	
    stRecipe.stUBL.lrDispencer1SuckValveOpenVolumeShow.lrDefault:=0;
	stRecipe.stUBL.lrDispencer1SuckValveOpenVolumeShow.lrMinLimit:=0;
	stRecipe.stUBL.lrDispencer1SuckValveOpenVolumeShow.lrMaxLimit:=1000;
	
    stRecipe.stUBL.lrDispencer1SuckVelocityShow.lrDefault:=300;
	stRecipe.stUBL.lrDispencer1SuckVelocityShow.lrMinLimit:=1;
	stRecipe.stUBL.lrDispencer1SuckVelocityShow.lrMaxLimit:=10000;
	
    stRecipe.stUBL.lrDispencer2DoseSuckingTimeDelayShow.lrDefault:=0;
	stRecipe.stUBL.lrDispencer2DoseSuckingTimeDelayShow.lrMinLimit:=0;
	stRecipe.stUBL.lrDispencer2DoseSuckingTimeDelayShow.lrMaxLimit:=1000;
	
    stRecipe.stUBL.lrDispencer2DoseSuckingVolumeShow.lrDefault:=0;
	stRecipe.stUBL.lrDispencer2DoseSuckingVolumeShow.lrMinLimit:=0;
	stRecipe.stUBL.lrDispencer2DoseSuckingVolumeShow.lrMaxLimit:=1000;
	
    stRecipe.stUBL.lrDispencer2DoseValveCloseTimeDecShow.lrDefault:=0;
	stRecipe.stUBL.lrDispencer2DoseValveCloseTimeDecShow.lrMinLimit:=0;
	stRecipe.stUBL.lrDispencer2DoseValveCloseTimeDecShow.lrMaxLimit:=1000;
	
    stRecipe.stUBL.lrDispencer2DoseValveCloseVolumeShow.lrDefault:=1;
	stRecipe.stUBL.lrDispencer2DoseValveCloseVolumeShow.lrMinLimit:=0;
	stRecipe.stUBL.lrDispencer2DoseValveCloseVolumeShow.lrMaxLimit:=1000;
	
	stRecipe.stUBL.udiDispencer2DosingDoneDelayTimeShow.udiDefault:=0;
	stRecipe.stUBL.udiDispencer2DosingDoneDelayTimeShow.udiMinLimit:=0;
	stRecipe.stUBL.udiDispencer2DosingDoneDelayTimeShow.udiMaxLimit:=1000;
	
    stRecipe.stUBL.lrDispencer2DoseValveOpenTimeAccShow.lrDefault:=200;
	stRecipe.stUBL.lrDispencer2DoseValveOpenTimeAccShow.lrMinLimit:=0;
	stRecipe.stUBL.lrDispencer2DoseValveOpenTimeAccShow.lrMaxLimit:=1000;
	
    stRecipe.stUBL.lrDispencer2DoseVolumeShow.lrDefault:=495;
	stRecipe.stUBL.lrDispencer2DoseVolumeShow.lrMinLimit:=0;
	stRecipe.stUBL.lrDispencer2DoseVolumeShow.lrMaxLimit:=1000;
	
    stRecipe.stUBL.lrDispencer2LifterStartDosePositionShow.lrDefault:=80;
	stRecipe.stUBL.lrDispencer2LifterStartDosePositionShow.lrMinLimit:=-1000;
	stRecipe.stUBL.lrDispencer2LifterStartDosePositionShow.lrMaxLimit:=1000;	
	
    stRecipe.stUBL.lrDispencer2LifterStopDosePositionShow.lrDefault:=192;
	stRecipe.stUBL.lrDispencer2LifterStopDosePositionShow.lrMinLimit:=-1000;
	stRecipe.stUBL.lrDispencer2LifterStopDosePositionShow.lrMaxLimit:=1000;
	
    stRecipe.stUBL.lrDispencer2Phase1AccelerationShow.lrDefault:=600;
	stRecipe.stUBL.lrDispencer2Phase1AccelerationShow.lrMinLimit:=1;
	stRecipe.stUBL.lrDispencer2Phase1AccelerationShow.lrMaxLimit:=100000;
	
    stRecipe.stUBL.lrDispencer2Phase1DecelerationShow.lrDefault:=150;
	stRecipe.stUBL.lrDispencer2Phase1DecelerationShow.lrMinLimit:=1;
	stRecipe.stUBL.lrDispencer2Phase1DecelerationShow.lrMaxLimit:=100000;
	
    stRecipe.stUBL.lrDispencer2Phase1VelocityShow.lrDefault:=140;
	stRecipe.stUBL.lrDispencer2Phase1VelocityShow.lrMinLimit:=1;
	stRecipe.stUBL.lrDispencer2Phase1VelocityShow.lrMaxLimit:=10000;
	
    stRecipe.stUBL.lrDispencer2Phase1VolumeShow.lrDefault:=0;
	stRecipe.stUBL.lrDispencer2Phase1VolumeShow.lrMinLimit:=0;
	stRecipe.stUBL.lrDispencer2Phase1VolumeShow.lrMaxLimit:=1000;
	
    stRecipe.stUBL.lrDispencer2Phase2AccelerationShow.lrDefault:=400;
	stRecipe.stUBL.lrDispencer2Phase2AccelerationShow.lrMinLimit:=1;
	stRecipe.stUBL.lrDispencer2Phase2AccelerationShow.lrMaxLimit:=100000;	
	
    stRecipe.stUBL.lrDispencer2Phase2DecelerationShow.lrDefault:=2000;
	stRecipe.stUBL.lrDispencer2Phase2DecelerationShow.lrMinLimit:=1;
	stRecipe.stUBL.lrDispencer2Phase2DecelerationShow.lrMaxLimit:=100000;
	
    stRecipe.stUBL.lrDispencer2Phase2VelocityShow.lrDefault:=140;
	stRecipe.stUBL.lrDispencer2Phase2VelocityShow.lrMinLimit:=1;
	stRecipe.stUBL.lrDispencer2Phase2VelocityShow.lrMaxLimit:=10000;
	
    stRecipe.stUBL.lrDispencer2Phase2VolumeShow.lrDefault:=0;
	stRecipe.stUBL.lrDispencer2Phase2VolumeShow.lrMinLimit:=0;
	stRecipe.stUBL.lrDispencer2Phase2VolumeShow.lrMaxLimit:=10000;	
	
    stRecipe.stUBL.lrDispencer2Phase3AccelerationShow.lrDefault:=50;
	stRecipe.stUBL.lrDispencer2Phase3AccelerationShow.lrMinLimit:=1;
	stRecipe.stUBL.lrDispencer2Phase3AccelerationShow.lrMaxLimit:=100000;	
	
    stRecipe.stUBL.lrDispencer2Phase3DecelerationShow.lrDefault:=50;
	stRecipe.stUBL.lrDispencer2Phase3DecelerationShow.lrMinLimit:=1;
	stRecipe.stUBL.lrDispencer2Phase3DecelerationShow.lrMaxLimit:=100000;
	
    stRecipe.stUBL.lrDispencer2Phase3VelocityShow.lrDefault:=50;
	stRecipe.stUBL.lrDispencer2Phase3VelocityShow.lrMinLimit:=1;
	stRecipe.stUBL.lrDispencer2Phase3VelocityShow.lrMaxLimit:=10000;
	
    stRecipe.stUBL.lrDispencer2SuckAccelerationShow.lrDefault:=3000;
	stRecipe.stUBL.lrDispencer2SuckAccelerationShow.lrMinLimit:=1;
	stRecipe.stUBL.lrDispencer2SuckAccelerationShow.lrMaxLimit:=100000;
	
    stRecipe.stUBL.lrDispencer2SuckValveCloseTimeDelayShow.lrDefault:=0;
	stRecipe.stUBL.lrDispencer2SuckValveCloseTimeDelayShow.lrMinLimit:=0;
	stRecipe.stUBL.lrDispencer2SuckValveCloseTimeDelayShow.lrMaxLimit:=4000;
	
    stRecipe.stUBL.lrDispencer2SuckValveOpenTimeDelayShow.lrDefault:=0;
	stRecipe.stUBL.lrDispencer2SuckValveOpenTimeDelayShow.lrMinLimit:=0;
	stRecipe.stUBL.lrDispencer2SuckValveOpenTimeDelayShow.lrMaxLimit:=1000;
	
    stRecipe.stUBL.lrDispencer2SuckValveOpenVolumeShow.lrDefault:=0;
	stRecipe.stUBL.lrDispencer2SuckValveOpenVolumeShow.lrMinLimit:=0;
	stRecipe.stUBL.lrDispencer2SuckValveOpenVolumeShow.lrMaxLimit:=1000;
	
    stRecipe.stUBL.lrDispencer2SuckVelocityShow.lrDefault:=300;
	stRecipe.stUBL.lrDispencer2SuckVelocityShow.lrMinLimit:=1;
	stRecipe.stUBL.lrDispencer2SuckVelocityShow.lrMaxLimit:=10000;
	
    stRecipe.stUBL.lrDispencersCatch1ClosedValueShow.lrDefault:=23.5;
	stRecipe.stUBL.lrDispencersCatch1ClosedValueShow.lrMinLimit:=0;
	stRecipe.stUBL.lrDispencersCatch1ClosedValueShow.lrMaxLimit:=200000;
	
    stRecipe.stUBL.lrDispencersCatch1OpenValueShow.lrDefault:=66.7;
	stRecipe.stUBL.lrDispencersCatch1OpenValueShow.lrMinLimit:=0;
	stRecipe.stUBL.lrDispencersCatch1OpenValueShow.lrMaxLimit:=200000;
	
    stRecipe.stUBL.lrDispencersCatch2ClosedValueShow.lrDefault:=15.8;
	stRecipe.stUBL.lrDispencersCatch2ClosedValueShow.lrMinLimit:=0;
	stRecipe.stUBL.lrDispencersCatch2ClosedValueShow.lrMaxLimit:=200000;
	
    stRecipe.stUBL.lrDispencersCatch2OpenValueShow.lrDefault:=56.7;
	stRecipe.stUBL.lrDispencersCatch2OpenValueShow.lrMinLimit:=0;
	stRecipe.stUBL.lrDispencersCatch2OpenValueShow.lrMaxLimit:=200000;
	
    stRecipe.stUBL.lrDispencersCatch3ClosedValueShow.lrDefault:=17.6;
	stRecipe.stUBL.lrDispencersCatch3ClosedValueShow.lrMinLimit:=0;
	stRecipe.stUBL.lrDispencersCatch3ClosedValueShow.lrMaxLimit:=200000;
	
	stRecipe.stUBL.lrDispencersCatch3OpenValueShow.lrDefault:=58.5;
	stRecipe.stUBL.lrDispencersCatch3OpenValueShow.lrMinLimit:=0;
	stRecipe.stUBL.lrDispencersCatch3OpenValueShow.lrMaxLimit:=200000;
	
    stRecipe.stUBL.lrDispencersCatch4ClosedValueShow.lrDefault:=22.7;
	stRecipe.stUBL.lrDispencersCatch4ClosedValueShow.lrMinLimit:=0;
	stRecipe.stUBL.lrDispencersCatch4ClosedValueShow.lrMaxLimit:=200000;
	
    stRecipe.stUBL.lrDispencersCatch4OpenValueShow.lrDefault:=67;
	stRecipe.stUBL.lrDispencersCatch4OpenValueShow.lrMinLimit:=0;
	stRecipe.stUBL.lrDispencersCatch4OpenValueShow.lrMaxLimit:=200000;
	
    stRecipe.stUBL.lrDispencersCatchHeightSVShow.lrDefault:=215;
	stRecipe.stUBL.lrDispencersCatchHeightSVShow.lrMinLimit:=-500;
	stRecipe.stUBL.lrDispencersCatchHeightSVShow.lrMaxLimit:=1000;
	
    stRecipe.stUBL.lrDispencersCatchToleranceShow.lrDefault:=15;
	stRecipe.stUBL.lrDispencersCatchToleranceShow.lrMinLimit:=0;
	stRecipe.stUBL.lrDispencersCatchToleranceShow.lrMaxLimit:=200;
	
    stRecipe.stUBL.lrDispencersLifterReadyPositionShow.lrDefault:=280;
	stRecipe.stUBL.lrDispencersLifterReadyPositionShow.lrMinLimit:=-1000;
	stRecipe.stUBL.lrDispencersLifterReadyPositionShow.lrMaxLimit:=1000;
	
    stRecipe.stUBL.lrFormsDragingLeftAccelerationShow.lrDefault:=2400;
	stRecipe.stUBL.lrFormsDragingLeftAccelerationShow.lrMinLimit:=100;
	stRecipe.stUBL.lrFormsDragingLeftAccelerationShow.lrMaxLimit:=10000;
	
    stRecipe.stUBL.lrFormsDragingLeftDecelerationShow.lrDefault:=2400;
	stRecipe.stUBL.lrFormsDragingLeftDecelerationShow.lrMinLimit:=100;
	stRecipe.stUBL.lrFormsDragingLeftDecelerationShow.lrMaxLimit:=10000;
	
    stRecipe.stUBL.lrFormsDragingLeftVelocityShow.lrDefault:=500;
	stRecipe.stUBL.lrFormsDragingLeftVelocityShow.lrMinLimit:=100;
	stRecipe.stUBL.lrFormsDragingLeftVelocityShow.lrMaxLimit:=1000;
	
    stRecipe.stUBL.lrFormsDragingRightAccelerationShow.lrDefault:=2400;
	stRecipe.stUBL.lrFormsDragingRightAccelerationShow.lrMinLimit:=100;
	stRecipe.stUBL.lrFormsDragingRightAccelerationShow.lrMaxLimit:=10000;
	
    stRecipe.stUBL.lrFormsDragingRightDecelerationShow.lrDefault:=2400;
	stRecipe.stUBL.lrFormsDragingRightDecelerationShow.lrMinLimit:=100;
	stRecipe.stUBL.lrFormsDragingRightDecelerationShow.lrMaxLimit:=10000;
	
    stRecipe.stUBL.lrFormsDragingRightVelocityShow.lrDefault:=500;
	stRecipe.stUBL.lrFormsDragingRightVelocityShow.lrMinLimit:=100;
	stRecipe.stUBL.lrFormsDragingRightVelocityShow.lrMaxLimit:=1000;
	
    stRecipe.stUBL.lrGripperScrewer1FindingScrewDegreeShow.lrDefault:=260;
	stRecipe.stUBL.lrGripperScrewer1FindingScrewDegreeShow.lrMinLimit:=0;
	stRecipe.stUBL.lrGripperScrewer1FindingScrewDegreeShow.lrMaxLimit:=10000;
	
    stRecipe.stUBL.lrGripperScrewer1VelocityShow.lrDefault:=90;
	stRecipe.stUBL.lrGripperScrewer1VelocityShow.lrMinLimit:=0;
	stRecipe.stUBL.lrGripperScrewer1VelocityShow.lrMaxLimit:=100000;

    stRecipe.stUBL.lrGripperScrewerCatchPressureShow.lrDefault:=20;
	stRecipe.stUBL.lrGripperScrewerCatchPressureShow.lrMinLimit:=0;
	stRecipe.stUBL.lrGripperScrewerCatchPressureShow.lrMaxLimit:=100;
		
    stRecipe.stUBL.lrGripperScrewerPressureShow.lrDefault:=40;
	stRecipe.stUBL.lrGripperScrewerPressureShow.lrMinLimit:=0;
	stRecipe.stUBL.lrGripperScrewerPressureShow.lrMaxLimit:=100;
	
    stRecipe.stUBL.lrGripperScrewerPushingCapPositionShow.lrDefault:=345;
	stRecipe.stUBL.lrGripperScrewerPushingCapPositionShow.lrMinLimit:=-10000;
	stRecipe.stUBL.lrGripperScrewerPushingCapPositionShow.lrMaxLimit:=10000;
	
    stRecipe.stUBL.lrGripperScrewerReadyPositionShow.lrDefault:=355;
	stRecipe.stUBL.lrGripperScrewerReadyPositionShow.lrMinLimit:=-100000;
	stRecipe.stUBL.lrGripperScrewerReadyPositionShow.lrMaxLimit:=100000;
	
    stRecipe.stUBL.lrGripperScrewerScrewingCapPositionShow.lrDefault:=345;
	stRecipe.stUBL.lrGripperScrewerScrewingCapPositionShow.lrMinLimit:=-10000;
	stRecipe.stUBL.lrGripperScrewerScrewingCapPositionShow.lrMaxLimit:=10000;
	
    stRecipe.stUBL.lrGripperScrewerThreadPitchShow.lrDefault:=0.5;
	stRecipe.stUBL.lrGripperScrewerThreadPitchShow.lrMinLimit:=0.1;
	stRecipe.stUBL.lrGripperScrewerThreadPitchShow.lrMaxLimit:=100;
	
    stRecipe.stUBL.lrGripperScrewerThreadTimesShow.lrDefault:=1;
	stRecipe.stUBL.lrGripperScrewerThreadTimesShow.lrMinLimit:=1;
	stRecipe.stUBL.lrGripperScrewerThreadTimesShow.lrMaxLimit:=4;
	
    stRecipe.stUBL.lrGripperScrewerTurnoversToFullScrewedShow.lrDefault:=0.5;
	stRecipe.stUBL.lrGripperScrewerTurnoversToFullScrewedShow.lrMinLimit:=0;
	stRecipe.stUBL.lrGripperScrewerTurnoversToFullScrewedShow.lrMaxLimit:=100;
	
    stRecipe.stUBL.lrGripperScrewing2TightTorqueShow.lrDefault:=1.1;
	stRecipe.stUBL.lrGripperScrewing2TightTorqueShow.lrMinLimit:=0;
	stRecipe.stUBL.lrGripperScrewing2TightTorqueShow.lrMaxLimit:=10;
	
    stRecipe.stUBL.lrGripperScrewingTightTorqueShow.lrDefault:=0.8;
	stRecipe.stUBL.lrGripperScrewingTightTorqueShow.lrMinLimit:=0;
	stRecipe.stUBL.lrGripperScrewingTightTorqueShow.lrMaxLimit:=10;
	
    stRecipe.stUBL.lrLidFeederDragingStationAccelerationShow.lrDefault:=2400;
	stRecipe.stUBL.lrLidFeederDragingStationAccelerationShow.lrMinLimit:=100;
	stRecipe.stUBL.lrLidFeederDragingStationAccelerationShow.lrMaxLimit:=10000;
	
    stRecipe.stUBL.lrLidFeederDragingStationDecelerationShow.lrDefault:=2400;
	stRecipe.stUBL.lrLidFeederDragingStationDecelerationShow.lrMinLimit:=100;
	stRecipe.stUBL.lrLidFeederDragingStationDecelerationShow.lrMaxLimit:=10000;
	
    stRecipe.stUBL.lrLidFeederDragingStationVelocityShow.lrDefault:=500;
	stRecipe.stUBL.lrLidFeederDragingStationVelocityShow.lrMinLimit:=100;
	stRecipe.stUBL.lrLidFeederDragingStationVelocityShow.lrMaxLimit:=10000;
	
    stRecipe.stUBL.lrLidFeederHeightPosSVShow.lrDefault:=309;
	stRecipe.stUBL.lrLidFeederHeightPosSVShow.lrMinLimit:=0;
	stRecipe.stUBL.lrLidFeederHeightPosSVShow.lrMaxLimit:=1000;
	
    stRecipe.stUBL.lrLidSealerDragingStationAccelerationShow.lrDefault:=2400;
	stRecipe.stUBL.lrLidSealerDragingStationAccelerationShow.lrMinLimit:=100;
	stRecipe.stUBL.lrLidSealerDragingStationAccelerationShow.lrMaxLimit:=10000;
	
    stRecipe.stUBL.lrLidSealerDragingStationDecelerationShow.lrDefault:=2400;
	stRecipe.stUBL.lrLidSealerDragingStationDecelerationShow.lrMinLimit:=100;
	stRecipe.stUBL.lrLidSealerDragingStationDecelerationShow.lrMaxLimit:=10000;
	
    stRecipe.stUBL.lrLidSealerDragingStationVelocityShow.lrDefault:=500;
	stRecipe.stUBL.lrLidSealerDragingStationVelocityShow.lrMinLimit:=100;
	stRecipe.stUBL.lrLidSealerDragingStationVelocityShow.lrMaxLimit:=1000;
	
    stRecipe.stUBL.lrLidSealerHeightPosSVShow.lrDefault:=285;
	stRecipe.stUBL.lrLidSealerHeightPosSVShow.lrMinLimit:=0;
	stRecipe.stUBL.lrLidSealerHeightPosSVShow.lrMaxLimit:=1000;
	
    stRecipe.stUBL.lrLidSealerPressureShow.lrDefault:=100;
	stRecipe.stUBL.lrLidSealerPressureShow.lrMinLimit:=0;
	stRecipe.stUBL.lrLidSealerPressureShow.lrMaxLimit:=1000;
	
    stRecipe.stUBL.lrWeightLowerToleranceShow.lrDefault:=1500;
	stRecipe.stUBL.lrWeightLowerToleranceShow.lrMinLimit:=1;
	stRecipe.stUBL.lrWeightLowerToleranceShow.lrMaxLimit:=10000;
	
    stRecipe.stUBL.lrWeightMassSVShow.lrDefault:=495;
	stRecipe.stUBL.lrWeightMassSVShow.lrMinLimit:=0;
	stRecipe.stUBL.lrWeightMassSVShow.lrMaxLimit:=1000;
	
    stRecipe.stUBL.lrWeightUpperToleranceShow.lrDefault:=1500;
	stRecipe.stUBL.lrWeightUpperToleranceShow.lrMinLimit:=1;
	stRecipe.stUBL.lrWeightUpperToleranceShow.lrMaxLimit:=10000;
	
    stRecipe.stUBL.nFormTransportersBeforeScrewerVelocitySVShow.udiDefault:=1100;
	stRecipe.stUBL.nFormTransportersBeforeScrewerVelocitySVShow.udiMinLimit:=0;
	stRecipe.stUBL.nFormTransportersBeforeScrewerVelocitySVShow.udiMaxLimit:=1500;
	
	stRecipe.stUBL.nBadBottleConveyorVelocitySVShow.udiDefault:=1200;
	stRecipe.stUBL.nBadBottleConveyorVelocitySVShow.udiMinLimit:=0;
	stRecipe.stUBL.nBadBottleConveyorVelocitySVShow.udiMaxLimit:=1500;
	
    stRecipe.stUBL.nFormTransportersDispencerVelocitySVShow.udiDefault:=1200;
	stRecipe.stUBL.nFormTransportersDispencerVelocitySVShow.udiMinLimit:=0;
	stRecipe.stUBL.nFormTransportersDispencerVelocitySVShow.udiMaxLimit:=1500;
	
    stRecipe.stUBL.nFormTransportersScrewerVelocitySVShow.udiDefault:=1200;
	stRecipe.stUBL.nFormTransportersScrewerVelocitySVShow.udiMinLimit:=0;
	stRecipe.stUBL.nFormTransportersScrewerVelocitySVShow.udiMaxLimit:=1500;
	
    stRecipe.stUBL.nGripperScrewer1TightTimeShow.diDefault:=100;
	stRecipe.stUBL.nGripperScrewer1TightTimeShow.diMinLimit:=0;
	stRecipe.stUBL.nGripperScrewer1TightTimeShow.diMaxLimit:=10000;
	
    stRecipe.stUBL.nGripperScrewerCatchHeightSVShow.diDefault:=160;
	stRecipe.stUBL.nGripperScrewerCatchHeightSVShow.diMinLimit:=0;
	stRecipe.stUBL.nGripperScrewerCatchHeightSVShow.diMaxLimit:=10000;
	
	stRecipe.stUBF.bBottleSorterBrushEnableShow.bDefault:=FALSE;
	stRecipe.stUBF.bBottleSorterHopperTransporterEnableShow.bDefault:=FALSE;
	stRecipe.stUBF.bBottleSorterRecieverEnableShow.bDefault:=FALSE;
	stRecipe.stUBF.bBottleSorterRecieverSlot1EnableShow.bDefault:=FALSE;
	stRecipe.stUBF.bBottleSorterRecieverSlot2EnableShow.bDefault:=FALSE;
	stRecipe.stUBF.bBottleSorterRecieverSlot3EnableShow.bDefault:=FALSE;
	stRecipe.stUBF.bBottleSorterRobotEnableShow.bDefault:=FALSE;
	stRecipe.stUBF.bBottleSorterSupplyTransporterEnableShow.bDefault:=FALSE;
	stRecipe.stUBF.bBottleSorterTransferTransporterEnableShow.bDefault:=FALSE;
	stRecipe.stUBF.bBottleSorterWeelEnableShow.bDefault:=FALSE;
	
	stRecipe.stUBF.iBottleSorterBrushEmptyingSpeedSVShow.diDefault:=10;
	stRecipe.stUBF.iBottleSorterBrushEmptyingSpeedSVShow.diMinLimit:=1;
    stRecipe.stUBF.iBottleSorterBrushEmptyingSpeedSVShow.diMaxLimit:=100;

	stRecipe.stUBF.iBottleSorterBrushRunningSpeedSVShow.diDefault:=10;
	stRecipe.stUBF.iBottleSorterBrushRunningSpeedSVShow.diMinLimit:=1;
	stRecipe.stUBF.iBottleSorterBrushRunningSpeedSVShow.diMaxLimit:=100;

	stRecipe.stUBF.iBottleSorterDistanceToFindElementOnSupplyConveyorDownstairsLimitSVShow.diDefault:=100;
	stRecipe.stUBF.iBottleSorterDistanceToFindElementOnSupplyConveyorDownstairsLimitSVShow.diMinLimit:=10;
	stRecipe.stUBF.iBottleSorterDistanceToFindElementOnSupplyConveyorDownstairsLimitSVShow.diMaxLimit:=10000;

	stRecipe.stUBF.iBottleSorterDistanceToFindElementOnTransferConveyorLimitEmptyingSVShow.diDefault:=100;
    stRecipe.stUBF.iBottleSorterDistanceToFindElementOnTransferConveyorLimitEmptyingSVShow.diMinLimit:=10;
	stRecipe.stUBF.iBottleSorterDistanceToFindElementOnTransferConveyorLimitEmptyingSVShow.diMaxLimit:=10000;

	stRecipe.stUBF.iBottleSorterDistanceToFindElementOnTransferConveyorLimitRunningSVShow.diDefault:=10;
    stRecipe.stUBF.iBottleSorterDistanceToFindElementOnTransferConveyorLimitRunningSVShow.diMinLimit:=1;
	stRecipe.stUBF.iBottleSorterDistanceToFindElementOnTransferConveyorLimitRunningSVShow.diMaxLimit:=100;

	stRecipe.stUBF.iBottleSorterHopperConveyorEmptyingSpeedSVShow.diDefault:=10;
    stRecipe.stUBF.iBottleSorterHopperConveyorEmptyingSpeedSVShow.diMinLimit:=1;
	stRecipe.stUBF.iBottleSorterHopperConveyorEmptyingSpeedSVShow.diMaxLimit:=100;

	stRecipe.stUBF.iBottleSorterHopperConveyorRunningSpeedSVShow.diDefault:=10;
    stRecipe.stUBF.iBottleSorterHopperConveyorRunningSpeedSVShow.diMinLimit:=1;
	stRecipe.stUBF.iBottleSorterHopperConveyorRunningSpeedSVShow.diMaxLimit:=100;

	stRecipe.stUBF.iBottleSorterSensorsCountFirstConditionSVShow.diDefault:=10;
    stRecipe.stUBF.iBottleSorterSensorsCountFirstConditionSVShow.diMinLimit:=0;
	stRecipe.stUBF.iBottleSorterSensorsCountFirstConditionSVShow.diMaxLimit:=1000;

	stRecipe.stUBF.iBottleSorterSensorsCountSecondConditionMaxSVShow.diDefault:=10;
    stRecipe.stUBF.iBottleSorterSensorsCountSecondConditionMaxSVShow.diMinLimit:=0;
	stRecipe.stUBF.iBottleSorterSensorsCountSecondConditionMaxSVShow.diMaxLimit:=1000;

	stRecipe.stUBF.iBottleSorterSupplyTimeFirstConditionSVShow.diDefault:=10;
    stRecipe.stUBF.iBottleSorterSupplyTimeFirstConditionSVShow.diMinLimit:=1;
	stRecipe.stUBF.iBottleSorterSupplyTimeFirstConditionSVShow.diMaxLimit:=10000;

	stRecipe.stUBF.iBottleSorterSupplyTimeSecondConditionSVShow.diDefault:=10;
    stRecipe.stUBF.iBottleSorterSupplyTimeSecondConditionSVShow.diMinLimit:=0;
	stRecipe.stUBF.iBottleSorterSupplyTimeSecondConditionSVShow.diMaxLimit:=1000;

	stRecipe.stUBF.iBottleSorterTransferConveyorEmptyingSpeedSVShow.diDefault:=10;
	stRecipe.stUBF.iBottleSorterTransferConveyorEmptyingSpeedSVShow.diMinLimit:=1;
	stRecipe.stUBF.iBottleSorterTransferConveyorEmptyingSpeedSVShow.diMaxLimit:=100;

	stRecipe.stUBF.iBottleSorterTransferConveyorRunningSpeedSVShow.diDefault:=10;
    stRecipe.stUBF.iBottleSorterTransferConveyorRunningSpeedSVShow.diMinLimit:=1;
	stRecipe.stUBF.iBottleSorterTransferConveyorRunningSpeedSVShow.diMaxLimit:=100;

	stRecipe.stUBF.lrBottleSorterBrushHeightPositionSVShow.lrDefault:=0;
	stRecipe.stUBF.lrBottleSorterBrushHeightPositionSVShow.lrMinLimit:=0;
	stRecipe.stUBF.lrBottleSorterBrushHeightPositionSVShow.lrMaxLimit:=100;

	stRecipe.stUBF.lrBottleSorterModuloMoveOffsetSVShow.lrDefault:=10;
	stRecipe.stUBF.lrBottleSorterModuloMoveOffsetSVShow.lrMinLimit:=1;
	stRecipe.stUBF.lrBottleSorterModuloMoveOffsetSVShow.lrMaxLimit:=360;

	stRecipe.stUBF.lrBottleSorterRecieverHeightPositionSVShow.lrDefault:=100;
    stRecipe.stUBF.lrBottleSorterRecieverHeightPositionSVShow.lrMinLimit:=10;
	stRecipe.stUBF.lrBottleSorterRecieverHeightPositionSVShow.lrMaxLimit:=200;

	stRecipe.stUBF.lrBottleSorterWheelEmptyingSpeedSVShow.lrDefault:=10;
    stRecipe.stUBF.lrBottleSorterWheelEmptyingSpeedSVShow.lrMinLimit:=5;
	stRecipe.stUBF.lrBottleSorterWheelEmptyingSpeedSVShow.lrMaxLimit:=100;

	stRecipe.stUBF.lrBottleSorterWheelSpeedSVShow.lrDefault:=10;
    stRecipe.stUBF.lrBottleSorterWheelSpeedSVShow.lrMinLimit:=5;
	stRecipe.stUBF.lrBottleSorterWheelSpeedSVShow.lrMaxLimit:=100;

	stRecipe.stUBF.uiBottleSorterSupplyTransporterEmptingSpeedSVShow.udiDefault:=100;
    stRecipe.stUBF.uiBottleSorterSupplyTransporterEmptingSpeedSVShow.udiMinLimit:=10;
	stRecipe.stUBF.uiBottleSorterSupplyTransporterEmptingSpeedSVShow.udiMaxLimit:=10000;

	stRecipe.stUBF.uiBottleSorterSupplyTransporterRunningSpeedSVShow.udiDefault:=100;
	stRecipe.stUBF.uiBottleSorterSupplyTransporterRunningSpeedSVShow.udiMinLimit:=10;
	stRecipe.stUBF.uiBottleSorterSupplyTransporterRunningSpeedSVShow.udiMaxLimit:=10000;
	
	stRecipe.stUBF.nBottleSorterRobotRecipeId.udiDefault:=70000;
	stRecipe.stUBF.nBottleSorterRobotRecipeId.udiMinLimit:=70000;
	stRecipe.stUBF.nBottleSorterRobotRecipeId.udiMaxLimit:=79999;
	
	stRecipe.stUCF.lrCapSorterBottleHightShow.lrDefault:=1;
	stRecipe.stUCF.lrCapSorterBottleHightShow.lrMinLimit:=1;
	stRecipe.stUCF.lrCapSorterBottleHightShow.lrMaxLimit:=1000;
	
	stRecipe.stUCF.lrCapSorterBottleNeckHightShow.lrDefault:=1;
	stRecipe.stUCF.lrCapSorterBottleNeckHightShow.lrMinLimit:=1;
	stRecipe.stUCF.lrCapSorterBottleNeckHightShow.lrMaxLimit:=1000;
	
	stRecipe.stUCF.lrCapSorterCapHightShow.lrDefault:=1;
	stRecipe.stUCF.lrCapSorterCapHightShow.lrMinLimit:=1;
	stRecipe.stUCF.lrCapSorterCapHightShow.lrMaxLimit:=1000;
	
	stRecipe.stUCF.lrCapSorterCapNeckHightShow.lrDefault:=1;
	stRecipe.stUCF.lrCapSorterCapNeckHightShow.lrMinLimit:=1;
	stRecipe.stUCF.lrCapSorterCapNeckHightShow.lrMaxLimit:=1000;
	
	stRecipe.stUCF.lrCapSorterPreScrewerPickerSpeedWhenScrewerShow.lrDefault:=10;
	stRecipe.stUCF.lrCapSorterPreScrewerPickerSpeedWhenScrewerShow.lrMinLimit:=5;
	stRecipe.stUCF.lrCapSorterPreScrewerPickerSpeedWhenScrewerShow.lrMaxLimit:=100;

	stRecipe.stUCF.LrCapSorterPreScrewerCheckStrawCatcherActuatorZPosition.lrDefault:=284;
	stRecipe.stUCF.LrCapSorterPreScrewerCheckStrawCatcherActuatorZPosition.lrMinLimit:=0;
	stRecipe.stUCF.LrCapSorterPreScrewerCheckStrawCatcherActuatorZPosition.lrMaxLimit:=1000;
	
	stRecipe.stUCF.bCapSorterBrush1OnWheelEnableShow.bDefault:=TRUE;
	stRecipe.stUCF.bCapSorterBrush2OnWheelEnableShow.bDefault:=FALSE;
	stRecipe.stUCF.bCapSorterCameraEnableShow.bDefault:=TRUE;
	stRecipe.stUCF.bCapSorterFeederEnableShow.bDefault:=TRUE;
	stRecipe.stUCF.bCapSorterFeederEnableTubeError.bDefault:=FALSE;
	stRecipe.stUCF.bCapSorterIntermediateBrushEnableShow.bDefault:=TRUE;
	stRecipe.stUCF.bCapSorterIntermediateTransporterEnableShow.bDefault:=TRUE;
    stRecipe.stUCF.bCapSorterPreScrewerBottleCatcherEnableShow.bDefault:=TRUE;
    stRecipe.stUCF.bCapSorterPreScrewerCatchAngleOpenEnaShow.bDefault:=FALSE;
    stRecipe.stUCF.bCapSorterPreScrewerEnableShow.bDefault:=TRUE;
    stRecipe.stUCF.bCapSorterPreScrewerPicker1EnableShow.bDefault:=TRUE;
    stRecipe.stUCF.bCapSorterPreScrewerPicker2EnableShow.bDefault:=TRUE;
    stRecipe.stUCF.bCapSorterPreScrewerPicker3EnableShow.bDefault:=TRUE;
    stRecipe.stUCF.bCapSorterPreScrewerPicker4EnableShow.bDefault:=TRUE;
    stRecipe.stUCF.bCapSorterPreScrewerPoundedInCap.bDefault:=FALSE;
    stRecipe.stUCF.bCapSorterRobotEnableShow.bDefault:=TRUE;
    stRecipe.stUCF.bCapSorterTransporterEnableShow.bDefault:=TRUE;
    stRecipe.stUCF.bCapSorterWheelEnableShow.bDefault:=TRUE;
    stRecipe.stUCF.bPresenceBottleEnableShow.bDefault:=FALSE;
	
	stRecipe.stUCF.iCapSorterBrush1OnWheelAutoSpeedShow.diDefault:=30;
	stRecipe.stUCF.iCapSorterBrush1OnWheelAutoSpeedShow.diMinLimit:=1;
	stRecipe.stUCF.iCapSorterBrush1OnWheelAutoSpeedShow.diMaxLimit:=100;
	
    stRecipe.stUCF.iCapSorterBrush1OnWheelEmptyingSpeedShow.diDefault:=30;
	stRecipe.stUCF.iCapSorterBrush1OnWheelEmptyingSpeedShow.diMinLimit:=1;
	stRecipe.stUCF.iCapSorterBrush1OnWheelEmptyingSpeedShow.diMaxLimit:=100;

    stRecipe.stUCF.iCapSorterBrush2OnWheelAutoSpeedShow.diDefault:=20;
	stRecipe.stUCF.iCapSorterBrush2OnWheelAutoSpeedShow.diMinLimit:=1;
	stRecipe.stUCF.iCapSorterBrush2OnWheelAutoSpeedShow.diMaxLimit:=100;
	
    stRecipe.stUCF.iCapSorterBrush2OnWheelEmptyingSpeedShow.diDefault:=30;
	stRecipe.stUCF.iCapSorterBrush2OnWheelEmptyingSpeedShow.diMinLimit:=1;
	stRecipe.stUCF.iCapSorterBrush2OnWheelEmptyingSpeedShow.diMaxLimit:=100;

    stRecipe.stUCF.iCapSorterIntermediateBrushAutoSpeedShow.diDefault:=60;
	stRecipe.stUCF.iCapSorterIntermediateBrushAutoSpeedShow.diMinLimit:=1;
	stRecipe.stUCF.iCapSorterIntermediateBrushAutoSpeedShow.diMaxLimit:=100;
	
    stRecipe.stUCF.iCapSorterIntermediateBrushEmptyingSpeedShow.diDefault:=30;
	stRecipe.stUCF.iCapSorterIntermediateBrushEmptyingSpeedShow.diMinLimit:=1;
	stRecipe.stUCF.iCapSorterIntermediateBrushEmptyingSpeedShow.diMaxLimit:=100;

    stRecipe.stUCF.iCapSorterIntermediateTransporterAutoSpeedShow.diDefault:=20;
	stRecipe.stUCF.iCapSorterIntermediateTransporterAutoSpeedShow.diMinLimit:=1;
	stRecipe.stUCF.iCapSorterIntermediateTransporterAutoSpeedShow.diMaxLimit:=100;
	
    stRecipe.stUCF.iCapSorterIntermediateTransporterDelayCountTimeShow.diDefault:=100;
	stRecipe.stUCF.iCapSorterIntermediateTransporterDelayCountTimeShow.diMinLimit:=0;
	stRecipe.stUCF.iCapSorterIntermediateTransporterDelayCountTimeShow.diMaxLimit:=100000;	
	
    stRecipe.stUCF.iCapSorterIntermediateTransporterEmptyingSpeedShow.diDefault:=100;
	stRecipe.stUCF.iCapSorterIntermediateTransporterEmptyingSpeedShow.diMinLimit:=1;
	stRecipe.stUCF.iCapSorterIntermediateTransporterEmptyingSpeedShow.diMaxLimit:=100;

	stRecipe.stUCF.iCapSorterIntermediateTransporterReverseTimeShow.diDefault:=4000;
	stRecipe.stUCF.iCapSorterIntermediateTransporterReverseTimeShow.diMinLimit:=0;
	stRecipe.stUCF.iCapSorterIntermediateTransporterReverseTimeShow.diMaxLimit:=10000;
	
    stRecipe.stUCF.iCapSorterProductType.diDefault:=0;
	stRecipe.stUCF.iCapSorterProductType.diMinLimit:=0;
	stRecipe.stUCF.iCapSorterProductType.diMaxLimit:=100;
	
    stRecipe.stUCF.iCapSorterRobotAccelerationDecelerationShow.diDefault:=20;
	stRecipe.stUCF.iCapSorterRobotAccelerationDecelerationShow.diMinLimit:=20;
	stRecipe.stUCF.iCapSorterRobotAccelerationDecelerationShow.diMaxLimit:=100;
	
    stRecipe.stUCF.iCapSorterRobotPickElevationShow.diDefault:=100;
	stRecipe.stUCF.iCapSorterRobotPickElevationShow.diMinLimit:=30;
	stRecipe.stUCF.iCapSorterRobotPickElevationShow.diMaxLimit:=1000;
	
    stRecipe.stUCF.iCapSorterRobotPickPositionZShow.diDefault:=16;
	stRecipe.stUCF.iCapSorterRobotPickPositionZShow.diMinLimit:=0;
	stRecipe.stUCF.iCapSorterRobotPickPositionZShow.diMaxLimit:=200;
	
    stRecipe.stUCF.iCapSorterRobotPickTimeShow.diDefault:=40;
	stRecipe.stUCF.iCapSorterRobotPickTimeShow.diMinLimit:=0;
	stRecipe.stUCF.iCapSorterRobotPickTimeShow.diMaxLimit:=10000;
	
    stRecipe.stUCF.iCapSorterRobotPlaceTimeShow.diDefault:=80;
	stRecipe.stUCF.iCapSorterRobotPlaceTimeShow.diMinLimit:=0;
	stRecipe.stUCF.iCapSorterRobotPlaceTimeShow.diMaxLimit:=1000;
	
    stRecipe.stUCF.iCapSorterRobotProductDiametr.diDefault:=20;
	stRecipe.stUCF.iCapSorterRobotProductDiametr.diMinLimit:=1;
	stRecipe.stUCF.iCapSorterRobotProductDiametr.diMaxLimit:=200;
	
    stRecipe.stUCF.iCapSorterRobotTCP_Lenght.diDefault:=30;
	stRecipe.stUCF.iCapSorterRobotTCP_Lenght.diMinLimit:=1;
	stRecipe.stUCF.iCapSorterRobotTCP_Lenght.diMaxLimit:=200;
	
    stRecipe.stUCF.iCapSorterRobotTCP_PlaceOffsetShow.diDefault:=1;
	stRecipe.stUCF.iCapSorterRobotTCP_PlaceOffsetShow.diMinLimit:=1;
	stRecipe.stUCF.iCapSorterRobotTCP_PlaceOffsetShow.diMaxLimit:=1000;
	
	stRecipe.stUCF.iCapSorterRobotVacuumActivationShow.diDefault:=60;
	stRecipe.stUCF.iCapSorterRobotVacuumActivationShow.diMinLimit:=0;
	stRecipe.stUCF.iCapSorterRobotVacuumActivationShow.diMaxLimit:=1000;
	
    stRecipe.stUCF.iCapSorterRobotVacuumOffShow.diDefault:=400;
	stRecipe.stUCF.iCapSorterRobotVacuumOffShow.diMinLimit:=0;
	stRecipe.stUCF.iCapSorterRobotVacuumOffShow.diMaxLimit:=1000;
	
    stRecipe.stUCF.iCapSorterTransporterEmptyingConveyorSpeedShow.diDefault:=25;
	stRecipe.stUCF.iCapSorterTransporterEmptyingConveyorSpeedShow.diMinLimit:=1;
	stRecipe.stUCF.iCapSorterTransporterEmptyingConveyorSpeedShow.diMaxLimit:=100;
	
    stRecipe.stUCF.iCapSorterTransporterStartDelayTimeShow.diDefault:=150;
	stRecipe.stUCF.iCapSorterTransporterStartDelayTimeShow.diMinLimit:=0;
	stRecipe.stUCF.iCapSorterTransporterStartDelayTimeShow.diMaxLimit:=10000;
	
    stRecipe.stUCF.iCapSorterTransporterTankConveyorVelocityShow.diDefault:=10;
	stRecipe.stUCF.iCapSorterTransporterTankConveyorVelocityShow.diMinLimit:=1;
	stRecipe.stUCF.iCapSorterTransporterTankConveyorVelocityShow.diMaxLimit:=100;
	
